OP10B_RH_ROTY(
	bAxis1_Ref_Switch:= , 
	bInit:= OP10_SRV_BLCK_INTZ , 
	bErrorReset:= Servo_Reset, 
	bEnable:= Servo_Enable , 
	bMoveVelocity:= , 
	bHalt:= , 
	bManualMode:= OP10B_MANUAL_SELECTED , 
	fHomePos:= , 
	fOverride:= , 
	fTargetPosition:= OP10B_SRV_RH_BDYANG_CNT.Position, 
	fTargetVelocity:= OP10_SERVO_POS_VEL_LIMIT.OP10B_RH_ROTRY_VELOCITY, 
	fAcc:= , 
	fDec:= , 
	Servo_High_Limit:= OP10_SERVO_POS_VEL_LIMIT.OP10B_RH_ROTRY_POS_LIMIT,
    Servo_Low_Limit:=OP10_SERVO_POS_VEL_LIMIT.OP10B_RH_ROTRY_NEG_LIMIT, 
	Safe_move_Conditions:= Servo_Safety,
	TORQUE_APPLIED :=  , 
	Axis:= OP10B_RH_ROTARY, 
	bHome:= OP10B_SRV_RH_BDYANG_CNT.Axis_Home_Cmd, 
	bSetPosition:= FESTO_NOT_NEED , 
	bMoveAbsolute:= OP10B_SRV_RH_BDYANG_CNT.ABSmove_Start, 
	bMoveRelative:= NOT_REQ , 
	bMoveTorque:= NOT_REQ , 
	stManualModeAxis:= OP10B_SRV_RH_BDYANG_STUS, 
	sAxisState=> OP10B_SRV_RH_BDYANG_CNT.Axis_State, 
	bAxis_ready=> , 
	bAxisInPosition=> , 
	bAxisError=> OP10B_SRV_RH_BDYANG_CNT.Axis_Error, 
	bAxisEnabled=> , 
	bAxisHomed=> , 
	bSetPositionDone=> , 
	bHaltDone=> , 
	bSTOPDone=> , 
	bHomeDone=> OP10B_SRV_RH_BDYANG_CNT.Axis_In_Home, 
	bDone=> , 
	bTorqueReached=> , 
	bsafe_to_move=> , 
	baxis_in_home_pos=> , 
	bABS_Pos_done=> OP10B_SRV_RH_BDYANG_CNT.Axis_In_Pos, 
	Actual_position=>,
	Actual_velocity=> , 
	Actual_Torque=> );
	
OP10B_LH_GRIPR(
	bAxis1_Ref_Switch:= , 
	bInit:= OP10_SRV_BLCK_INTZ , 
	bErrorReset:= Servo_Reset, 
	bEnable:= Servo_Enable , 
	bMoveVelocity:= , 
	bHalt:= , 
	bManualMode:= OP10B_MANUAL_SELECTED , 
	fHomePos:= , 
	fOverride:= , 
	fTargetPosition:= OP10B_SRV_LH_BDYGRP_CNT.Position, 
	fTargetVelocity:= OP10_SERVO_POS_VEL_LIMIT.OP10B_LH_GRPR_VELOCITY, 
	fAcc:= , 
	fDec:= ,
	Servo_High_Limit:= OP10_SERVO_POS_VEL_LIMIT.OP10B_LH_GRPR_POS_LIMIT,
    Servo_Low_Limit:=OP10_SERVO_POS_VEL_LIMIT.OP10B_LH_GRPR_NEG_LIMIT,  
	Safe_move_Conditions:= Servo_Safety,
	TORQUE_APPLIED := , 
	Axis:= OP10B_LH_GRIPPER, 
	bHome:= OP10B_SRV_LH_BDYGRP_CNT.Axis_Home_Cmd, 
	bSetPosition:= FESTO_NOT_NEED , 
	bMoveAbsolute:= OP10B_SRV_LH_BDYGRP_CNT.ABSmove_Start, 
	bMoveRelative:= NOT_REQ , 
	bMoveTorque:= NOT_REQ , 
	stManualModeAxis:= OP10B_SRV_LH_BDYGRP_STUS, 
 	sAxisState=> OP10B_SRV_LH_BDYGRP_CNT.Axis_State, 
	bAxis_ready=> , 
	bAxisInPosition=> , 
	bAxisError=> OP10B_SRV_LH_BDYGRP_CNT.Axis_Error, 
	bAxisEnabled=> , 
	bAxisHomed=> , 
	bSetPositionDone=> , 
	bHaltDone=> , 
	bSTOPDone=> , 
	bHomeDone=> OP10B_SRV_LH_BDYGRP_CNT.Axis_In_Home, 
	bDone=> , 
	bTorqueReached=> , 
	bsafe_to_move=> , 
	baxis_in_home_pos=> , 
	bABS_Pos_done=> OP10B_SRV_LH_BDYGRP_CNT.Axis_In_Pos , 
	Actual_position=>, 
	Actual_velocity=> , 
	Actual_Torque=> );
	
OP10B_RH_GRIPR(
	bAxis1_Ref_Switch:= , 
	bInit:= OP10_SRV_BLCK_INTZ , 
	bErrorReset:= Servo_Reset, 
	bEnable:= Servo_Enable  , 
	bMoveVelocity:= , 
	bHalt:= , 
	bManualMode:= OP10B_MANUAL_SELECTED , 
	fHomePos:= , 
	fOverride:= , 
	fTargetPosition:= OP10B_SRV_RH_BDYGRP_CNT.Position, 
	fTargetVelocity:= OP10_SERVO_POS_VEL_LIMIT.OP10B_RH_GRPR_VELOCITY, 
	fAcc:= , 
	fDec:= ,
	Servo_High_Limit:= OP10_SERVO_POS_VEL_LIMIT.OP10B_RH_GRPR_POS_LIMIT,
    Servo_Low_Limit:=OP10_SERVO_POS_VEL_LIMIT.OP10B_RH_GRPR_NEG_LIMIT, 
	Safe_move_Conditions:=Servo_Safety,
	TORQUE_APPLIED := , 
	Axis:= OP10B_RH_GRIPPER, 
	bHome:= OP10B_SRV_RH_BDYGRP_CNT.Axis_Home_Cmd, 
	bSetPosition:= FESTO_NOT_NEED , 
	bMoveAbsolute:= OP10B_SRV_RH_BDYGRP_CNT.ABSmove_Start, 
	bMoveRelative:= NOT_REQ , 
	bMoveTorque:= NOT_REQ , 
	stManualModeAxis:= OP10B_SRV_RH_BDYGRP_STUS, 
 	sAxisState=> OP10B_SRV_RH_BDYGRP_CNT.Axis_State, 
	bAxis_ready=> , 
	bAxisInPosition=>, 
	bAxisError=> OP10B_SRV_RH_BDYGRP_CNT.Axis_Error, 
	bAxisEnabled=> , 
	bAxisHomed=> , 
	bSetPositionDone=> , 
	bHaltDone=> , 
	bSTOPDone=> , 
	bHomeDone=> OP10B_SRV_RH_BDYGRP_CNT.Axis_In_Home,  
	bDone=> , 
	bTorqueReached=> , 
	bsafe_to_move=> , 
	baxis_in_home_pos=> , 
	bABS_Pos_done=>  OP10B_SRV_RH_BDYGRP_CNT.Axis_In_Pos , 
	Actual_position=>, 
	Actual_velocity=> , 
	Actual_Torque=> );
	
	
OP10B_CONVEYOR(
	bAxis1_Ref_Switch:= , 
	bInit:= , 
	bErrorReset:= Servo_Reset , 
	bEnable:= Servo_Enable, 
	bMoveVelocity:=OP10B_SRV_O_CNVY_CNT.VELmove_Start, 
	bHalt:= , 
	bManualMode:= OP10B_MANUAL_SELECTED, 
	fHomePos:= , 
	fOverride:= , 
	fTargetPosition:=OP10B_SRV_O_CNVY_CNT.Position , 
	fTargetVelocity:=OP10B_SRV_O_CNVY_CNT.Velocity , 
	fAcc:= , 
	fDec:= , 
	Safe_move_Conditions:= Servo_Safety, 
	Axis:= OP10B_CONVRY, 
	HME_WRITE_ADD:= 16#5003,	
	bHome:= OP10B_SRV_O_CNVY_CNT.Bsethome , 
	bSetPosition:= OP10B_SRV_O_CNVY_CNT.BsetPos, 
	bMoveAbsolute:= OP10B_SRV_O_CNVY_CNT.ABSmove_Start, 
	bMoveRelative:= OP10B_SRV_O_CNVY_CNT.RELmove_Start, 
	bMoveTorque:= OP10B_SRV_O_CNVY_CNT.Torque_mode_Start, 
	stManualModeAxis:= OP10B_SRV_O_CNVY_STUS, 
	bmove_home:= OP10B_SRV_O_CNVY_CNT.Axis_Home_Cmd, 
	sAxisState=>OP10B_SRV_O_CNVY_CNT.Axis_State , 
	bAxis_ready=>OP10B_SRV_O_CNVY_CNT.Axis_ready , 
	bAxisInPosition=> , 
	bAxisError=> OP10B_SRV_O_CNVY_CNT.Axis_Error, 
	bAxisEnabled=> , 
	bAxisHomed=> , 
	bSetPositionDone=> , 
	bHaltDone=> , 
	bSTOPDone=> , 
	bHomeDone=> OP10B_SRV_O_CNVY_CNT.Axis_In_Home, 
	bDone=> , 
	bTorqueReached=> , 
	bsafe_to_move=> , 
	baxis_in_home_pos=> , 
	bABS_Pos_done=> , 
	Actual_position=> , 
	Actual_velocity=> , 
	Actual_Torque=> );
	
	   OP10A_SRV_RH_BDYANG_STUS.targetVelocity	:= 20;//OP10A_TARGET_VEL	
	   OP10A_SRV_LH_BDYANG_STUS.targetVelocity	:= 20;//OP10A_TARGET_VEL	
	   OP10A_SRV_RH_BDYGRP_STUS.targetVelocity	:= 20;//OP10A_TARGET_VEL	
	   OP10A_SRV_LH_BDYGRP_STUS.targetVelocity	:= 20;//OP10A_TARGET_VEL	
	   OP10A_SRV_LH_BDYGRP_STUS.targetVelocity	:= 20;//OP10A_TARGET_VEL	
	
	   OP10B_SRV_RH_BDYANG_STUS.targetVelocity	:= 20;//OP10B_TARGET_VEL	
	   OP10B_SRV_LH_BDYANG_STUS.targetVelocity	:= 20;//OP10B_TARGET_VEL	
	   OP10B_SRV_RH_BDYGRP_STUS.targetVelocity	:= 20;//OP10B_TARGET_VEL	
	   OP10B_SRV_LH_BDYGRP_STUS.targetVelocity	:= 20;//OP10B_TARGET_VEL	
	   OP10B_SRV_LH_BDYGRP_STUS.targetVelocity	:= 20;//OP10B_TARGET_VEL	
	
	
		OP10_SRV_FRST_PCKBDY_STUS.TARgetVelocity:=50;
		OP10_SRV_SCND_PCKBDY_STUS.TARgetVelocity:=50;

END_PROGRAM

// ---- FB/In_Range.TcPOU
FUNCTION In_Range : BOOL
VAR_INPUT
	value,setvalue,tolerance:LREAL;
END_VAR
VAR
	low: LREAL:= setvalue-tolerance;
	high:LREAL:= setvalue+tolerance;;
END_VAR

IF (value>=low) AND (value<=high) THEN
	In_Range:=TRUE;
ELSE
	In_Range:=FALSE;
END_IF

END_FUNCTION

// ---- POUs/Programs/OP10/OP10_HOMING.TcPOU
PROGRAM OP10_HOMING
VAR
	OP10A_ERR_TMR				: TON;
	OP10B_ERR_TMR				: TON;
	OP10A_ROBO_RST_SEQ			: INT;	
	OP10B_ROBO_RST_SEQ			: INT;
	OP10A_START_HOMING			: BOOL;
	OP10B_START_HOMING			: BOOL;
	OP10A_ROBO_INZI_DN			: BOOL;	
	OP10B_ROBO_INZI_DN			: BOOL;	
	temp_42						: BOOL;	
	temp_43						: BOOL;	
END_VAR

//#############################		OP10	###########################################

IF (OP10A_START_HOMNG OR OP10B_START_HOMNG) AND (NOT (OP10A_AUTO_RUNNING OR OP10A_STEP_RUNNING OR OP10B_AUTO_RUNNING OR OP10B_STEP_RUNNING OR 
	 OP10A_Rbt_In_Pick_Zone OR OP10B_Rbt_In_Pick_Zone)) THEN
	OP10_A_SRV_SCND_BDYPCK_HME		:= (OP10_BDY_SING_FRT.Sensor1 AND OP10_BDY_SING_SEC.Sensor1) OR OP10_COMP_PICKED_1;		
	OP10_A_SRV_FST_BDYPCK_HME	    := (OP10_BDY_SING_FRT.Sensor1 AND OP10_BDY_SING_SEC.Sensor1) OR OP10_COMP_PICKED_2;
	OP10_FRT_CYL_INITZAL			:= NOT OP10_COMP_PICKED_1;
	OP10_SEC_CYL_INITZAL			:= NOT OP10_COMP_PICKED_2;	
END_IF

//#############################		OP10A	################################

R1(CLK:= OP10A_START_HOMING AND NOT OP10A_ERR AND NOT OP10A_AUTO_RUNNING AND NOT OP10A_STEP_RUNNING, Q=> );
IF R1.Q THEN
	OP10A_START_HOMNG		:= TRUE;
	OP10A_START_HOMING		:= FALSE;
	OP10A_HME_STP_NO		:= 1;
	OP10A_ROBO_RST_SEQ		:= 0;
	OP10_COMP_PICKED_1		:= 0;	// need to be deleted
	OP10_COMP_PICKED_2		:= 0;
	OP10A_Sing_Seq			:=10;
	OP10B_Sing_Seq			:=10;	
END_IF
IF OP10A_ALL_HOME OR OP10A_ERR THEN
	OP10A_START_HOMNG		:= FALSE;	
END_IF

IF (OP10A_HME_STP_NO = 10) AND OP10A_START_HOMNG THEN
	OP10A_ROBO_SFE_HME		:= TRUE;
IF OP10A_Rbt_In_Home THEN
	OP10A_HME_STP_NO 		:= OP10A_HME_10_15;
END_IF
END_IF

OP10A_ALL_HOME	:= OP10_SRV_FRST_PCKBDY_HME_FB AND OP10_SRV_SCND_PCKBDY_HME_FB AND OP10A_Rbt_In_Home AND 
					(OP10A_HME_STP_NO=30)AND (OP10A_ROBO_RST_SEQ=30) AND OP10A_GRIPPER_HOME AND ((OP10_BDY_SING_FRT.Sensor1 OR OP10_COMP_PICKED_1)AND 
						(OP10_BDY_SING_SEC.Sensor1 OR OP10_COMP_PICKED_2));



//####################################		OP10A_ROBO	RST		#################################

IF OP10A_START_HOMNG THEN
CASE OP10A_ROBO_RST_SEQ OF 
	
	0: 	OP10A_ROBO_MODE_NO				:= 3;	
		OP10A_ROBO_PRGM_RST				:= TRUE;
		OP10A_ROBO_RST_SEQ				:= 5;
		
	5:	IF (OP10A_ROBO_PRGM_RST =TRUE) AND (NOT OP10A_Program_Execute) THEN
		IF NOT OP10A_CMP_PRS_ROBO THEN
		OP10A_Homing_Start				:= TRUE;
		OP10A_ROBO_RST_SEQ				:= 10;
		ELSE
		OP10A_Homing_Start				:= TRUE;
		OP10A_PLACE_IN_REJECTION		:= TRUE;
		OP10A_ROBO_RST_SEQ				:= 100;	
		END_IF		
		OP10A_ROBO_PRGM_RST				:= FALSE;		
		END_IF	
	
	10: IF OP10A_Rbt_In_Home THEN
		OP10A_Homing_Start				:= FALSE;
		OP10A_ROBO_RST_SEQ				:= 15;
		END_IF

	15: IF OP10A_Rbt_In_Home THEN
		OP10A_Homing_Start				:= FALSE;
		OP10A_ROBO_MODE_NO				:= 1;
		OP10A_ROBO_PRGM_RST				:= TRUE;
		OP10A_ROBO_RST_SEQ				:= 20;			
		END_IF

	20: IF (OP10A_ROBO_MODE_NO=1) AND OP10A_ROBO_PRGM_RST AND NOT OP10A_Program_Execute THEN
		OP10A_ROBO_PRGM_RST				:= FALSE;
		OP10A_ROBO_RST_SEQ				:= 30;		
		END_IF

	100: IF OP10A_Rbt_In_Reject_Zone AND OP10A_ROBO_Gripper_Open THEN
		OP10A_PLACE_IN_REJECTION		:= FALSE;
		OP10A_ROBO_RST_SEQ				:= 15;
		 END_IF
END_CASE
END_IF

//#############################		OP10B	################################

R2(CLK:= OP10B_START_HOMING AND NOT OP10B_ERR AND NOT OP10B_AUTO_RUNNING AND NOT OP10B_STEP_RUNNING, Q=> );
IF R2.Q THEN
	OP10B_START_HOMNG		:= TRUE;
	OP10B_START_HOMING		:= FALSE;
	OP10B_HME_STP_NO		:= 1;
	OP10B_ROBO_RST_SEQ		:= 0;
	OP10_COMP_PICKED_1		:= 0;	// need to be deleted
	OP10_COMP_PICKED_2		:= 0;
	OP10A_Sing_Seq			:=10;
	OP10B_Sing_Seq			:=10;	
END_IF
IF OP10B_ALL_HOME OR OP10B_ERR THEN
	OP10B_START_HOMNG		:= FALSE;	
END_IF

IF (OP10B_HME_STP_NO = 10) AND OP10B_START_HOMNG THEN
	OP10B_ROBO_SFE_HME	:= TRUE;
IF OP10B_Rbt_In_Home THEN
	OP10B_HME_STP_NO := OP10B_HME_10_15;
END_IF
END_IF

OP10B_ALL_HOME	:= OP10_SRV_FRST_PCKBDY_HME_FB AND OP10_SRV_SCND_PCKBDY_HME_FB AND OP10B_Rbt_In_Home AND 
					(OP10B_HME_STP_NO=30) AND (OP10B_ROBO_RST_SEQ=30)AND OP10B_GRIPPER_HOME AND ((OP10_BDY_SING_FRT.Sensor1 OR OP10_COMP_PICKED_1)AND 
						(OP10_BDY_SING_SEC.Sensor1 OR OP10_COMP_PICKED_2)); 



//####################################		OP10B_ROBO	RST		#################################

IF OP10B_START_HOMNG THEN
CASE OP10B_ROBO_RST_SEQ OF 
	
	0:	OP10B_ROBO_MODE_NO				:= 3;	
		OP10B_ROBO_PRGM_RST				:= TRUE;
		OP10B_ROBO_RST_SEQ				:= 5;
		
	5:	IF (OP10B_ROBO_PRGM_RST =TRUE) AND (NOT OP10B_Program_Execute) THEN
		IF NOT OP10B_CMP_PRS_ROBO THEN
		OP10B_Homing_Start				:= TRUE;
		OP10B_ROBO_RST_SEQ				:= 10;
		ELSE
		OP10B_Homing_Start				:= TRUE;
		OP10B_PLACE_IN_REJECTION		:= TRUE;
		OP10B_ROBO_RST_SEQ				:= 100;	
		END_IF		
		OP10B_ROBO_PRGM_RST				:= FALSE;		
		END_IF	
	
	10: IF OP10B_Rbt_In_Home THEN
		OP10B_Homing_Start				:= FALSE;
		OP10B_ROBO_RST_SEQ				:= 15;
		END_IF

	15: IF OP10B_Rbt_In_Home THEN
		OP10B_Homing_Start				:= FALSE;
		OP10B_ROBO_MODE_NO				:= 1;
		OP10B_ROBO_PRGM_RST				:= TRUE;
		OP10B_ROBO_RST_SEQ				:= 20;			
		END_IF

	20: IF (OP10B_ROBO_MODE_NO=1) AND OP10B_ROBO_PRGM_RST AND NOT OP10B_Program_Execute THEN
		OP10B_ROBO_PRGM_RST				:= FALSE;
		OP10B_ROBO_RST_SEQ				:= 30;		
		END_IF

	100: IF OP10B_Rbt_In_Reject_Zone AND OP10B_ROBO_Gripper_Open THEN
		OP10B_PLACE_IN_REJECTION		:= FALSE;
		OP10B_ROBO_RST_SEQ				:= 15;
		 END_IF
END_CASE	
END_IF

END_PROGRAM

// ---- POUs/Programs/OP10/OP10A_AUTO.TcPOU
PROGRAM OP10A_AUTO
VAR	
	OP10A_ROBO_SYSTEM				: FB_Robot;
	OP10A_CYL_IP					: OP10_ORNG_CYL_IP;
	OP10A_CYL_OP					: OP10_ORNG_CYL_OP;
	OP10A_PNP_FB					: OP10_ORING_PNP;
	OP10A_ROBO_PNP_FB				: OP10_ROBO_PNP;
	OP10A_STN_MOVER					: INT;
	OP10A_OUT_ORNG_DN				: BOOL;
	OP10A_AGLE_LH_CMR_TRG			: BOOL;
	OP10A_AGLE_RH_CMR_TRG			: BOOL;	
	OP10A_RDY_TO_PLC_ORNG			: BOOL;
	OP10A_STN_ENABLE				: BOOL;
// TEMPERY


	OP10A_ROBO_MANUAL: BOOL;
	ORING_DN: BOOL;
	tmr: Ton;
	OP10A_PROCESS_DN: BOOL;
	OP10A_PROCESS_DN_: BOOL;
	
	OP10A_PROCESS_DN_TRG: R_TRIG;
	

END_VAR

VAR PERSISTENT
	OP10A_RESULT_UPDATE		: INT;
	OP10A_DELAY_TMR			: OP10_ORNG_CYL_DLY;
AFT_DEG_HME_DLY: TIME;	AFT_DEG_WRK_DLY: TIME;
	AFT_GRP_HME_DLY: TIME;
	AFT_GRP_WRK_DELY: TIME;
	AFT_HORZ_FRW_DELY: TIME;
END_VAR

OP10A_PNP_FB(
	AUTO:= OP10A_AUTO_RUNNING OR OP10A_STEP_RUNNING, 
	MANUAL:= OP10A_MANUAL_SELECTED, 
	ERROR:= OP10A_ERR, 
	START_ENABLE:= OP10A_START_ENABLE, 
	ROBO_MVED_SFE:= NOT OP10A_Rbt_In_O_Ring_Zone, 
	LH_CMR_OK:= OP10A_LH_CMR_OK AND OP10A_ORNG_RDY_PCK, 
	LH_CMR_NOK:= OP10A_LH_CMR_NOK AND OP10A_ORNG_RDY_PCK, 
	RH_CMR_OK:= OP10A_RH_CMR_OK AND OP10A_ORNG_RDY_PCK, 
	RH_CMR_NOK:= OP10A_RH_CMR_NOK AND OP10A_ORNG_RDY_PCK, 
	ROBO_REACHED:= OP10A_RDY_TO_PLC_ORNG, 
	CYL_INPUTS:= OP10A_CYL_IP, 
	DELY_TIME:= OP10A_DELAY_TMR,
	CONTINOUS_CHECK := OP10A_CYL_PNP_CHECK, 
	O_RING_PLCED=> OP10A_OUT_ORNG_DN, 
	RDY_TO_PICK_ORNG=> OP10A_CYL_RDY_TO_PLC, 
	LH_REJ_DONE=> , 
	RH_REJ_DONE=> , 
	CYL_OUTPUTS=> OP10A_CYL_OP,
	ORNG_PCK_FRM_CNVY := OP10A_ORNG_PCK_DN);

	
	
	
// OP10A AUTO LOGIC CYLINDERS MAPPING 

									(*SENSOR_I/P*)
	OP10A_CYL_IP.DEGREE_0				:=I10A_ORING_ROTRY_CYL_O_DEG_I1011_0;
	OP10A_CYL_IP.DEGREE_180				:=I10A_ORING_ROTRY_CYL_180_DEG_I1011_1;
    OP10A_CYL_IP.HORIZ_CYL_SNR1         :=I10A_ORING_HORZ_CYL_REV_I1011_2;
    OP10A_CYL_IP.HORIZ_CYL_SNR2         :=I10A_ORING_HORZ_CYL_FWD_I1011_3;
    OP10A_CYL_IP.LH_O_GRP_SNR1       	:=I10A_ORING_LH_GRPR_CLSE_I1010_2;
    OP10A_CYL_IP.LH_O_GRP_SNR2          :=I10A_ORING_LH_GRPR_OPN_I1010_3; 
    OP10A_CYL_IP.LH_O_PUSH_SNR1         := NOT I10A_ORING_LH_PUSHR_CYL_REV_I1010_4;
    OP10A_CYL_IP.LH_O_PUSH_SNR2         :=I10A_ORING_LH_PUSHR_CYL_REV_I1010_4;
    OP10A_CYL_IP.LH_REJ_SNR1            :=I10A_LH_FIRTRE_ORING_REJ_CYL_REV_I1011_6;
    OP10A_CYL_IP.LH_REJ_SNR2            :=I10A_LH_FIRTRE_ORING_REJ_CYL_FWD_I1011_7;
	OP10A_CYL_IP.RH_O_GRP_SNR1			:=I10A_ORING_RH_GRPR_CLSE_I1010_6;
    OP10A_CYL_IP.RH_O_GRP_SNR2          :=I10A_ORING_RH_GRPR_OPN_I1010_5;
    OP10A_CYL_IP.RH_O_PUSH_SNR1         := NOT I10A_ORING_RH_PUSHR_CYL_REV_I1010_7;
    OP10A_CYL_IP.RH_O_PUSH_SNR2         :=I10A_ORING_RH_PUSHR_CYL_REV_I1010_7;
    OP10A_CYL_IP.RH_REJ_SNR1            :=I10A_RH_FIRTRE_ORING_REJ_CYL_REV_I1020_0;
    OP10A_CYL_IP.RH_REJ_SNR2            :=I10A_RH_FIRTRE_ORING_REJ_CYL_FWD_I1020_1;
    OP10A_CYL_IP.VERT_CYL_SNR1          :=I10A_ORING_VERT_CYL_UP_I1011_4;
    OP10A_CYL_IP.VERT_CYL_SNR2          :=I10A_ORING_VERT_CYL_DWN_I1011_5;
	
									(*CYLINDER_AUTO_O/P*)	
	
	OP10A_ALL_CYL_HOME_FB				:=OP10A_CYL_OP.ALL_HOME			  ;
	OP10A_O_0DEGRE_AUTOCMD1				:=OP10A_CYL_OP.DEGREE_AUT_CMD1	  ;
	OP10A_O_180DEGRE_AUTOCMD2   		:=OP10A_CYL_OP.DEGREE_AUT_CMD2    ;
	OP10A_O_HORZ_AUTOCMD1    			:=OP10A_CYL_OP.HORIZ_CYL_AUT_CMD1 ;
	OP10A_O_HORZ_AUTOCMD2    			:=OP10A_CYL_OP.HORIZ_CYL_AUT_CMD2 ;
	OP10A_A_O_LHGRIP_ONOFF    			:=OP10A_CYL_OP.LH_O_GRP_VALVE_ON  ;
	OP10A_A_O_LHPUSH_CYL    			:=OP10A_CYL_OP.LH_O_PSH_VALVE_ON  ;
	OP10A_A_O_RHGRIP_ONOFF    			:=OP10A_CYL_OP.RH_O_GRP_VALVE_ON  ;
	OP10A_A_O_RHPUSH_CYL    			:=OP10A_CYL_OP.RH_O_PSH_VALVE_ON  ;
	OP10A_O_VERT_AUTOCMD1    			:=OP10A_CYL_OP.VERT_CYL_AUT_CMD1  ;
	OP10A_O_VERT_AUTOCMD2    			:=OP10A_CYL_OP.VERT_CYL_AUT_CMD2  ;

// 								DELAY_TIMER_FOR_CYLINDER

	OP10A_DELAY_TMR.AFT_DEG_HME_DLY		:= AFT_DEG_HME_DLY;
	OP10A_DELAY_TMR.AFT_DEG_WRK_DLY		:= AFT_DEG_WRK_DLY;
	OP10A_DELAY_TMR.AFT_GRP_HME_DLY		:= AFT_GRP_HME_DLY;
	OP10A_DELAY_TMR.AFT_GRP_WRK_DELY	:= AFT_GRP_WRK_DELY;
	OP10A_DELAY_TMR.AFT_HORZ_FRW_DELY	:= AFT_HORZ_FRW_DELY;
	







	
	
//###############		ROBO	################### 

OP10A_ROBO_PNP_FB(
	AUTO:= OP10A_AUTO_RUNNING OR OP10A_STEP_RUNNING, 
	MANUAL:= OP10A_MANUAL_SELECTED, 
	ERROR:= OP10A_ERR, 
	START_ENABLE:= OP10A_START_ENABLE, 
	ROBO_STATUS_FB:= OP10A_ROBO_STATUS, 
	ROBO_GRP_STUS:= OP10A_GRP_STATUS, 
	BDY1_RDY_PCK:= OP10_LH_CMP_RDY_PCK, 
	BDY2_RDY_PCK:= OP10_RH_CMP_RDY_PCK, 
	BDY1_PCK_BYPAS:= OP10A_BDY1_PCK_BYPAS, 
	BDY2_PCK_BYPAS:= OP10A_BDY2_PCK_BYPAS, 
	O_RNG_NEED:= , 
	PLC_OUTR_ORNG_DN:= OP10A_OUT_ORNG_DN OR ORING_DN, // DELETE ORING_DN
	CMR_RESULT_DN:= OP10A_CMR_DN_RSLT, 
	LH_CMR_ORNG_OK:= OP10A_LH_CMR_OK, 
	RH_CMR_ORING_OK:= OP10A_RH_CMR_OK,
	STN_ENABLE := OP10A_STN_ENABLE,
	OP10_STN_MOVER := OP10A_STN_MOVER,
	START_HOMING := OP10A_START_HOMNG,
	ROBO_IN_HOME := OP10A_Rbt_In_Home,
	STN_MOVER_NUM := OP10A_STN_MOVER,
	LH_BODY_GRIP_HME_DN := OP10A_SRV_LH_BDYGRP_CNT.Axis_In_Home,
	RH_BODY_GRIP_HME_DN := OP10A_SRV_RH_BDYGRP_CNT.Axis_In_Home,
	LH_BODY_ROTRY_HME_DN := OP10A_SRV_LH_BDYANG_CNT.Axis_In_Home,
	RH_BODY_ROTRY_HME_DN := OP10A_SRV_RH_BDYANG_CNT.Axis_In_Home,
	SEC_SING_CYL_SNR1 := OP10_BDY_SING_SEC.Sensor1,
	FRT_SING_CYL_SNR1 := OP10_BDY_SING_FRT.Sensor1,
	CMP_GRIPPED := OP10A_CMP_PRS_ROBO,
	ROBO_GRP_OPN := OP10A_ROBO_Gripper_Open,
	ROBO_IN_ORING_ZONE := OP10A_Rbt_In_O_Ring_Zone,
	ROBO_CTRL_WRD=> OP10A_ROBO_CNTRL, 
	ROBO_GRP_CNTRL=> OP10A_GRP_CNTRL, 
	LH_CAMERA_TRIGGER=> OP10A_AGLE_LH_CMR_TRG, 
	RH_CAMERA_TRIGGER=> OP10A_AGLE_RH_CMR_TRG, 
	PLC_OUTR_ORNG=> OP10A_RDY_TO_PLC_ORNG,
	LH_PART_STATUS => ,
	RH_PART_STATUS => ,
	PROCESS_DONE => ,
	GRIPPER_HOME => OP10A_GRIPPER_HOME,
	OP10_CURR_MOVER => OP10A_CURR_MOVER,
	PROCESS_DONE := OP10A_PROCESS_DN);


	//OP10A_CMR_DN_RSLT			:= TRUE;						// should be deleted
	//OP10A_LH_CMR_OK             := TRUE;						// should be deleted
	//OP10A_RH_CMR_OK             := TRUE;						// should be deleted	


(*tmr(IN:= OP10A_STN_ENABLE, PT:=T#10MS , Q=> , ET=> );
	IF tmr.Q THEN
	IF (MOVER_CMP_STATUS[OP10A_STN_MOVER][1]=0) THEN
	MOVER_CMP_STATUS[OP10A_STN_MOVER][1] := 10;		
	END_IF
	IF (MOVER_CMP_STATUS[OP10A_STN_MOVER][2]=0) THEN
	MOVER_CMP_STATUS[OP10A_STN_MOVER][2] := 10;
	END_IF	
	ALL_STATION_DONE.POSITION_DONE[OP10A_XTS_POS_NO]:= TRUE;
	END_IF*)
	
	CASE OP10A_RESULT_UPDATE OF
		0: IF OP10A_PROCESS_DN THEN
			OP10A_RESULT_UPDATE			:= 5;
		END_IF
		
		5: 	IF OP10A_PROCESS_DN THEN
			IF (MOVER_CMP_STATUS[OP10A_STN_MOVER][1]=0) THEN
			MOVER_CMP_STATUS[OP10A_CURR_MOVER][1] := OP10A_ROBO_PNP_FB.LH_PART_STATUS;		
			END_IF
			IF (MOVER_CMP_STATUS[OP10A_STN_MOVER][2]=0) THEN
			MOVER_CMP_STATUS[OP10A_CURR_MOVER][2] := OP10A_ROBO_PNP_FB.RH_PART_STATUS;
			END_IF		
			IF OP10A_PROCESS_DN AND (OP10A_CURR_MOVER = OP10A_STN_MOVER) AND (MOVER_CMP_STATUS[OP10A_STN_MOVER][1]=10 OR MOVER_CMP_STATUS[OP10A_STN_MOVER][1]=11) AND 
		(MOVER_CMP_STATUS[OP10A_STN_MOVER][2]=10 OR MOVER_CMP_STATUS[OP10A_STN_MOVER][2]=11) THEN
			OP10A_RESULT_UPDATE			:= 10;
			END_IF
			END_IF
	
		10:	STATION_DONE[OP10A_CURR_MOVER][OP10A_XTS_POS_NO]			:= TRUE;
			IF 	MOVER_STP_NO[OP10A_CURR_MOVER]<>((OP10A_XTS_POS_NO*10)+1)THEN
			OP10A_CURR_MOVER											:= 0;	
			OP10A_PROCESS_DN											:= FALSE;
			OP10A_RESULT_UPDATE											:= 15;
			END_IF
			
		15: OP10A_PROCESS_DN_TRG(CLK:= OP10A_PROCESS_DN, Q=> );
			IF OP10A_PROCESS_DN_TRG.Q THEN
			OP10A_RESULT_UPDATE											:= 0;	
			END_IF
	END_CASE
	

(*	IF OP10A_PROCESS_DN OR tmr.Q THEN
	IF (MOVER_CMP_STATUS[OP10A_STN_MOVER][1]=0) THEN
	MOVER_CMP_STATUS[OP10A_CURR_MOVER][1] := OP10A_ROBO_PNP_FB.LH_PART_STATUS;		
	END_IF
	IF (MOVER_CMP_STATUS[OP10A_STN_MOVER][2]=0) THEN
	MOVER_CMP_STATUS[OP10A_CURR_MOVER][2] := OP10A_ROBO_PNP_FB.RH_PART_STATUS;
	END_IF	
	END_IF
	IF OP10A_PROCESS_DN AND (OP10A_CURR_MOVER = OP10A_STN_MOVER) AND (MOVER_CMP_STATUS[OP10A_STN_MOVER][1]=10 OR MOVER_CMP_STATUS[OP10A_STN_MOVER][1]=11) AND 
		(MOVER_CMP_STATUS[OP10A_STN_MOVER][2]=10 OR MOVER_CMP_STATUS[OP10A_STN_MOVER][2]=11) THEN
	STATION_DONE[OP10A_CURR_MOVER][OP10A_XTS_POS_NO]			:= TRUE;
	IF 	MOVER_STP_NO[OP10A_CURR_MOVER]<>((OP10A_XTS_POS_NO*10)+1)THEN
	OP10A_CURR_MOVER											:= 0;	
	OP10A_PROCESS_DN											:= FALSE;	
	END_IF
	END_IF*)
// #############################		OP10A_ROBO_STATUS_CONTROL		#################################
	
	OP10A_ROBO_STATUS.BDY_PCK_POSITION	  		:= OP10A_ROBO_Gripper_Close AND OP10A_Rbt_In_Pick_Zone;//OP10A_Rbt_In_Pick_Zone
//	OP10A_ROBO_STATUS.BDY_S_PCK_POSITION		:= ;
	OP10A_ROBO_STATUS.BDY_CMR_CHK_POS		  	:= OP10A_Camera_Trigger; 							
//	OP10A_ROBO_STATUS.BDY_S_ORNG_POS		   	:= ;
	OP10A_ROBO_STATUS.BDY_ORNG_PLC_POS	  		:= OP10A_O_Ring_Pick_Pos_Reached AND OP10A_Rbt_In_O_Ring_Zone;//OP10A_Rbt_In_O_Ring_Zone
	OP10A_ROBO_STATUS.BDY_MVE_PLC_POS		  	:= OP10A_ROBO_Gripper_Open;//OP10A_Rbt_In_Place_Zone	
	OP10A_ROBO_STATUS.ROBO_SAFE_POS		    	:=  NOT OP10A_Rbt_In_Place_Zone;
	OP10A_ROBO_STATUS.ROBO_REJ_POS				:= OP10A_Rbt_In_Reject_Zone;

	OP10A_A_BODY_READY_TO_PICK					:= 	OP10A_ROBO_CNTRL.BDY_PCK_POSITION	;	
//	                                      	 	:=  OP10A_ROBO_CNTRL.BDY_S_PCK_POSITION;	    
	OP10A_A_PICK_PART_OK                   		:=  OP10A_ROBO_CNTRL.BDY_CMR_CHK_POS		;
//					                      		:= 	OP10A_ROBO_CNTRL.BDY_S_ORNG_POS		;    
	OP10A_A_CAMERA_OK                      		:= 	OP10A_ROBO_CNTRL.BDY_ORNG_PLC_POS OR OP10A_ROBO_CNTRL.BDY_MVE_PLC_POS;    
//	                                       		:= 	OP10A_ROBO_CNTRL.ROBO_SAFE_POS		;    
//	                                       		:= 	OP10A_ROBO_CNTRL.ROBO_REJ_POS		;   


// #############################		OP10A_GRIPPER_STATUS_CONTROL		#################################

	OP10A_GRP_STATUS.LH_BDY_GRP_WRK_FB			:= OP10A_A_SRV_LH_GRPWRK_FB	;
	OP10A_GRP_STATUS.LH_BDY_GRP_HOM_FB		    := OP10A_A_SRV_LH_GRPHME_FB	;
	OP10A_GRP_STATUS.RH_BDY_GRP_WRK_FB		    := OP10A_A_SRV_RH_GRPWRK_FB	;
	OP10A_GRP_STATUS.RH_BDY_GRP_HME_FB		    := OP10A_A_SRV_RH_GRPHME_FB	;
	OP10A_GRP_STATUS.LH_BDY_ROTRY_WRK_FB		:= OP10A_SRV_LH_BDYANG_WRK_FB;
	OP10A_GRP_STATUS.LH_BDY_ROTRY_HOM_FB		:= OP10A_SRV_LH_BDYANG_HME_FB;
	OP10A_GRP_STATUS.RH_BDY_ROTRY_WRK_FB		:= OP10A_SRV_RH_BDYANG_WRK_FB;
	OP10A_GRP_STATUS.RH_BDY_ROTRY_HME_FB		:= OP10A_SRV_RH_BDYANG_HME_FB;
	OP10A_GRP_STATUS.RH_BDY_ROTRY_ZERO_FB		:= OP10A_SRV_RH_BDYANG_ZERO_FB;
	OP10A_GRP_STATUS.LH_BDY_ROTRY_ZERO_FB		:= OP10A_SRV_LH_BDYANG_ZERO_FB;	
	OP10A_GRP_STATUS.RH_BDY_ROTRY_CMR_FB		:= OP10A_SRV_RH_BDYANG_CMR_FB;
	OP10A_GRP_STATUS.RH_BDY_RTRY_FITEE_FB		:= OP10A_SRV_RH_BDYANG_FITRE_FB;
	OP10A_GRP_STATUS.LH_BDY_ROTRY_CMR_FB		:= OP10A_SRV_LH_BDYANG_CMR_FB;	
	OP10A_GRP_STATUS.LH_BDY_RTRY_FITEE_FB		:= OP10A_SRV_LH_BDYANG_FITRE_FB;

	OP10A_A_SRV_LH_GRPWRK						:= OP10A_GRP_CNTRL.LH_BODY_GRIP_WRK	;
	OP10A_A_SRV_LH_GRPHME	        			:= OP10A_GRP_CNTRL.LH_BODY_GRIP_HOM;
	OP10A_A_SRV_RH_GRPWRK	        			:= OP10A_GRP_CNTRL.RH_BODY_GRIP_WRK	;  
	OP10A_A_SRV_RH_GRPHME	        			:= OP10A_GRP_CNTRL.RH_BODY_GRIP_HME	;
	OP10A_SRV_LH_BDYANG_WRK	        			:= OP10A_GRP_CNTRL.LH_BODY_ROTRY_WRK;	
	OP10A_SRV_LH_BDYANG_HME	        			:= OP10A_GRP_CNTRL.LH_BODY_ROTRY_HOM ;	
	OP10A_SRV_RH_BDYANG_WRK	        			:= OP10A_GRP_CNTRL.RH_BODY_ROTRY_WRK;	
	OP10A_SRV_RH_BDYANG_HME	        			:= OP10A_GRP_CNTRL.RH_BODY_ROTRY_HME ;	
	OP10A_SRV_LH_BDYANG_CMR						:= OP10A_GRP_CNTRL.LH_BODY_ROTRY_CMR;
	OP10A_SRV_LH_BDYANG_FITRE					:= OP10A_GRP_CNTRL.LH_BODY_RTRY_FITEE;	
	OP10A_SRV_RH_BDYANG_CMR						:= OP10A_GRP_CNTRL.RH_BODY_ROTRY_CMR;
	OP10A_SRV_RH_BDYANG_FITRE					:= OP10A_GRP_CNTRL.RH_BODY_RTRY_FITEE;
	
// STEPPER_NEGATIVE_HOME_METHOD
	                                               
	OP10A_SRV_LH_BDYGRP_CNT.Axis_Home_Cmd		:= OP10A_GRP_CNTRL.LH_BODY_GRIP_HOMING_1 ; 
	OP10A_SRV_RH_BDYGRP_CNT.Axis_Home_Cmd		:= OP10A_GRP_CNTRL.RH_BODY_GRIP_HOMING_1 ; 
	OP10A_SRV_LH_BDYANG_CNT.Axis_Home_Cmd		:= OP10A_GRP_CNTRL.LH_BODY_ROTRY_HOMING_1; 		
	OP10A_SRV_RH_BDYANG_CNT.Axis_Home_Cmd		:= OP10A_GRP_CNTRL.RH_BODY_ROTRY_HOMING_1; 
	
	
//#####################################	ROBO_FB	####################################


OP10A_ROBO_SYSTEM(
	i_b_Operation_Enable_Feedback:= OP10A_Auto_Operation_Enable, 
	i_b_Auto_Enable_Feedback:= OP10A_Mirror_Auto_enable, 
	i_b_Servo_On_Feedback:= OP10A_Servo_ON_OFF_Status, 
	i_b_Servo_Off_Feedback:= OP10A_Mirror_SRVO_Off, 
	i_b_Error_Feedback:= OP10A_H_Error OR OP10A_L_Error, 
	i_b_Program_Start_Enable_Feedback:= OP10A_Program_Execute, 
	i_b_Robo_Stopping_Feedback:= OP10A_Program_Waiting, 
	i_b_Emergency_Pressed_Feedback:= OP10A_During_EMG_Stop, 
	i_b_Auto_Mode_Feedback:= OP10A_Mirror_Auto_enable, 
	i_b_Reset:= Servo_Reset, 
	i_b_RobotAutoManual:= OP10A_AUTO_SELECTED OR OP10A_STEP_SELECTED OR OP10A_MANUAL_SELECTED, 
	i_b_ProgramReset:= OP10A_ROBO_PRGM_RST, 
	o_b_Operation_Enable_Cmd=> OP10A_Operation_Enable, 
	o_b_Auto_Enable_Cmd=> OP10A_Auto_Enable, 
	o_b_Servo_On_Cmd=> OP10A_Servo_ON, 
	o_b_Servo_Off_Cmd=> OP10A_SERVO_OFF, 
	o_b_Error_Reset_Cmd=> OP10A_ERR_RST, 
	o_b_Program_Reset_Cmd=> OP10A_PRGM_RST, 
	o_b_Program_Start_Cmd=> OP10A_Start, 
	o_b_Program_Stop_Cmd=> OP10A_Stop , 
	o_b_RobotAutoManual=> , 
	o_b_Error=> );	
	
	OP10A_STOP2					:=OP10A_Stop;
	WITH_ORING_VARIIENT			:= TRUE;				// NEED TO BE CHECKED FOR NOT ORING VARIENT 
	

//##############################			ROBO		#####################################

	IF (MANUAL_SELECTED AND OP10A_M_BODY_READY_TO_PICK) OR 
		(OP10A_A_BODY_READY_TO_PICK AND NOT OP10B_BODY_READY_TO_PICK AND NOT OP10B_Rbt_In_Pick_Zone) THEN
		OP10A_BODY_READY_TO_PICK						:= TRUE;// BODY COMPONENT READY;
		OP10A_Pick_Zone_Safe							:= (OP10A_A_SRV_LH_GRPHME_FB OR OP10A_BDY1_PCK_BYPAS) AND 
															(OP10A_A_SRV_RH_GRPHME_FB OR OP10A_BDY2_PCK_BYPAS ) AND 
 																OP10_LH_CMP_RDY_PCK AND OP10_RH_CMP_RDY_PCK; 
	ELSE
		OP10A_BODY_READY_TO_PICK						:= FALSE;
		OP10A_Pick_Zone_Safe							:= FALSE;					
	END_IF

	IF (MANUAL_SELECTED AND OP10A_M_PICK_PART_OK) OR OP10A_A_PICK_PART_OK THEN
		OP10A_PICK_PART_OK								:= TRUE;
		OP10A_A_ORING_INSERTION_DONE					:= TRUE;
		OP10A_Gripper_Rotate_Complete					:= TRUE;
		OP10A_Camera_Zone_Safe							:= TRUE;(*(OP10A_SRV_RH_BDYANG_CMR_FB OR OP10A_BDY2_PCK_BYPAS) AND 
															(OP10A_SRV_LH_BDYANG_CMR_FB OR OP10A_BDY1_PCK_BYPAS);*)
	ELSE
		OP10A_PICK_PART_OK								:= FALSE;
		OP10A_Gripper_Rotate_Complete					:= FALSE;
		OP10A_Camera_Zone_Safe							:= FALSE;
		OP10A_A_ORING_INSERTION_DONE					:= FALSE;		
	END_IF

	IF (MANUAL_SELECTED AND OP10A_M_PICK_PART_NOK) OR OP10A_A_PICK_PART_NOK THEN
		OP10A_PICK_PART_NOK								:= TRUE;
	ELSE
		OP10A_PICK_PART_NOK								:= FALSE;		
	END_IF

	IF (MANUAL_SELECTED AND OP10A_M_CAMERA_OK) OR OP10A_A_CAMERA_OK THEN
		OP10A_READY_TO_INSERT_ORING						:= TRUE;
		OP10A_Place_Zone_Safe							:= (OP10A_SRV_LH_BDYANG_WRK_FB OR OP10A_BDY1_PCK_BYPAS) AND 
															(OP10A_SRV_RH_BDYANG_WRK_FB OR OP10A_BDY2_PCK_BYPAS);
		OP10A_ROTATION_COMPLETE							:= TRUE;
		OP10A_O_Ring_Zone_Safe							:=  (OP10A_SRV_LH_BDYANG_FITRE_FB OR OP10A_BDY1_PCK_BYPAS) AND 
															(OP10A_SRV_RH_BDYANG_FITRE_FB OR OP10A_BDY2_PCK_BYPAS) AND 
																OP10A_CYL_RDY_TO_PLC;
		IF OP10A_ROBO_CNTRL.BDY_MVE_PLC_POS	THEN
		OP10A_A_PLACE_IN_CONVEYOR						:= TRUE;
		END_IF
		
		IF OP10A_Camera_Trigger THEN
		OP10A_CAMERA_OK									:= TRUE;	
		END_IF												
			
	ELSE                                            	
		OP10A_CAMERA_OK									:= FALSE;
		OP10A_READY_TO_INSERT_ORING						:= FALSE;
		OP10A_O_Ring_Zone_Safe							:= FALSE;
		OP10A_Place_Zone_Safe							:= FALSE;
		OP10A_A_PLACE_IN_CONVEYOR						:= FALSE;
		OP10A_ROTATION_COMPLETE							:= FALSE;		
	END_IF

	IF (MANUAL_SELECTED AND OP10A_M_CAMERA_NOK) OR OP10A_A_CAMERA_NOK AND OP10A_Camera_Trigger THEN
		OP10A_CAMERA_NOK								:= TRUE;
	ELSE
		OP10A_CAMERA_NOK								:= FALSE;		
	END_IF	    	 
              
 	IF (MANUAL_SELECTED AND OP10A_M_ORING_INSERTION_DONE) OR OP10A_A_ORING_INSERTION_DONE THEN
		OP10A_ORING_INSERTION_DONE						:= TRUE;
	ELSE
		OP10A_ORING_INSERTION_DONE						:= FALSE;		
	END_IF 
   
  	IF (MANUAL_SELECTED AND OP10A_M_PLACE_IN_CONVEYOR) OR OP10A_A_PLACE_IN_CONVEYOR THEN
		OP10A_PLACE_IN_CONVEYOR							:= TRUE;
	ELSE
		OP10A_PLACE_IN_CONVEYOR							:= FALSE;		
	END_IF
   
	OP10A_GRIPPER_OPEN									:= (OP10A_A_SRV_LH_GRPHME_FB OR OP10A_BDY1_PCK_BYPAS )AND (OP10A_A_SRV_RH_GRPHME_FB OR OP10A_BDY2_PCK_BYPAS) AND NOT OP10A_ROBO_Gripper_Close;
	OP10A_GRIPPER_CLOSE									:= (OP10A_A_SRV_LH_GRPWRK_FB OR OP10A_BDY1_PCK_BYPAS)AND (OP10A_A_SRV_RH_GRPWRK_FB OR OP10A_BDY2_PCK_BYPAS) AND OP10A_ROBO_Gripper_Close;

	OP10A_Reject_Zone_Safe								:= NOT OP10B_Rbt_In_Reject_Zone;








//############################		OP10A STATION ENABLE CONDITION		##########################

	OP10A_STN_MOVER					:= MOVER_POSITION[OP10A_XTS_POS_NO];
	IF AUTO_WITH_XTS THEN	
	IF OP10A_STN_MOVER>0 THEN
	IF NOT END_OF_CYCLE THEN
	OP10A_STN_ENABLE				:= MOVER_POS_RECHED[OP10A_STN_MOVER] AND ((MOVER_CMP_STATUS[OP10A_STN_MOVER][1]=0)OR 
										(MOVER_CMP_STATUS[OP10A_STN_MOVER][2]=0)) AND STATION_ENABLE_CONTROL AND NOT 
											(I10A_BDY1_PRSN_MOVER_I1001_3 OR I10A_BDY2_PRSN_MOVER_I1001_4);
	ELSE
	MOVER_CMP_STATUS[OP10A_STN_MOVER][1]					:=5;
	MOVER_CMP_STATUS[OP10A_STN_MOVER][2]					:=5;
	STATION_DONE[OP10A_STN_MOVER][OP10A_XTS_POS_NO]			:= TRUE;
	
	END_IF
	ELSE
	OP10A_STN_ENABLE										:= FALSE;	
	END_IF	
	END_IF

END_PROGRAM

// ---- FB/Robot/FB_Robot.TcPOU
FUNCTION_BLOCK FB_Robot
VAR_INPUT
	
	i_b_Operation_Enable_Feedback 		: BOOL;				// IO Enabled Feedback		
	i_b_Auto_Enable_Feedback 			: BOOL;				// Auto Enabled Feedback
	i_b_Servo_On_Feedback 				: BOOL;				// Servo On Feedback		
	i_b_Servo_Off_Feedback 				: BOOL;				// Servo Off Feedback		
	i_b_Error_Feedback					: BOOL;				// Error Feedback		
	i_b_Program_Start_Enable_Feedback 	: BOOL;				// Program Start Enable		
	i_b_Robo_Stopping_Feedback 			: BOOL;				// Robo Stopping Feedback		          		 
	i_b_Emergency_Pressed_Feedback 		: BOOL;				// Emergency Pressed Feedback		
	i_b_Auto_Mode_Feedback 				: BOOL;				// Auto Mode Feedback		bRoboAutoManual

	i_b_Reset							: BOOL;
	i_b_RobotAutoManual					: BOOL;
	i_b_ProgramReset					: BOOL;
	
END_VAR
VAR_OUTPUT
	
	o_b_Operation_Enable_Cmd 			: BOOL;				// IO Enable Command
	o_b_Auto_Enable_Cmd					: BOOL;				// Auto Enable Command
	o_b_Servo_On_Cmd					: BOOL;				// Servo On Command		
	o_b_Servo_Off_Cmd					: BOOL;				// Servo Off Command		
	o_b_Error_Reset_Cmd					: BOOL;				// Error Reset Command	
	o_b_Program_Reset_Cmd				: BOOL;				// Program Reset Command
	o_b_Program_Start_Cmd				: BOOL;				// Program Start Command					
	o_b_Program_Stop_Cmd				: BOOL;				// Program Stop Command	
	
	o_b_RobotAutoManual					: BOOL;
	o_b_Error							: BOOL;
END_VAR

VAR

	iState								: E_State_RobotGeneral;
	tonStateTimeOut						: TON;
	tonAutoManual						: ton;
	bRobotAutoManual					: BOOL;
	
	
END_VAR		

VAR_TEMP
	
	bTIN								: BOOL;	
	bTIN2								: BOOL;
	
END_VAR

	// Auto Manual
	o_b_RobotAutoManual:= i_b_Auto_Enable_Feedback AND NOT bRobotAutoManual;

CASE iState OF 
	

E_State_RobotGeneral.Init:

		o_b_Operation_Enable_Cmd	:= FALSE;
		o_b_Auto_Enable_Cmd			:= false;
		o_b_Servo_On_Cmd			:= false;
		o_b_Servo_Off_Cmd			:= false;
		o_b_Error_Reset_Cmd			:= false;
		o_b_Program_Reset_Cmd		:= false;
		o_b_Program_Start_Cmd		:= false;
		o_b_Program_Stop_Cmd		:= FALSE;
		
		IF i_b_ProgramReset THEN
			iState:=E_State_RobotGeneral.ProgramReset;
		ELSIF NOT i_b_Auto_Enable_Feedback THEN
			iState:=E_State_RobotGeneral.AutoEnable;	
		END_IF

E_State_RobotGeneral.AutoEnable:

		o_b_Operation_Enable_Cmd	:= FALSE;
		o_b_Auto_Enable_Cmd			:= TRUE;
		o_b_Servo_On_Cmd			:= false;
		o_b_Servo_Off_Cmd			:= false;
		o_b_Error_Reset_Cmd			:= false;
		o_b_Program_Reset_Cmd		:= false;
		o_b_Program_Start_Cmd		:= false;
		o_b_Program_Stop_Cmd		:= FALSE;

		bTIN:= i_b_RobotAutoManual;//TRUE;

		IF i_b_ProgramReset THEN
			iState:=E_State_RobotGeneral.ProgramReset;		
		ELSIF i_b_Auto_Enable_Feedback AND i_b_RobotAutoManual THEN
			bTIN:= FALSE;
			iState:=E_State_RobotGeneral.OperationEnable;
		ELSIF tonStateTimeOut.Q THEN 
			bTIN:= FALSE;
			iState:=E_State_RobotGeneral.Init;
		END_IF
		
		tonStateTimeOut(IN:=bTIN,PT:=T#1S);

E_State_RobotGeneral.OperationEnable:

		o_b_Operation_Enable_Cmd	:= TRUE;

		bTIN:= i_b_RobotAutoManual;//TRUE;

		IF i_b_ProgramReset THEN
			iState:=E_State_RobotGeneral.ProgramReset;		
		ELSIF  i_b_Error_Feedback THEN
			bTIN:= FALSE;
			iState:=E_State_RobotGeneral.Error;
		ELSIF NOT i_b_RobotAutoManual THEN
			bTIN:= FALSE;
			iState:=E_State_RobotGeneral.AutoEnable;
		ELSIF i_b_Operation_Enable_Feedback OR i_b_Auto_Enable_Feedback THEN
			bTIN:= FALSE;
			iState:=E_State_RobotGeneral.ServoOn;
		ELSIF tonStateTimeOut.Q THEN 
			bTIN:= FALSE;
			iState:=E_State_RobotGeneral.Error;
		END_IF
		
		tonStateTimeOut(IN:=bTIN,PT:=T#1S);

E_State_RobotGeneral.Error:

		o_b_Operation_Enable_Cmd	:= FALSE;
		o_b_Auto_Enable_Cmd			:= TRUE;
		o_b_Servo_On_Cmd			:= FALSE;
		o_b_Servo_Off_Cmd			:= false;
		o_b_Error_Reset_Cmd			:= false;
		o_b_Program_Reset_Cmd		:= false;
		o_b_Program_Start_Cmd		:= false;
		o_b_Program_Stop_Cmd		:= FALSE;

		IF i_b_ProgramReset THEN
			iState:=E_State_RobotGeneral.ProgramReset;
		ELSIF i_b_reset THEN
		iState:=E_State_RobotGeneral.ErrorReset;	
		END_IF
		
E_State_RobotGeneral.ErrorReset:

		o_b_Auto_Enable_Cmd			:= TRUE;
		o_b_Servo_On_Cmd			:= FALSE;
		o_b_Servo_Off_Cmd			:= false;
		o_b_Error_Reset_Cmd			:= TRUE;
		o_b_Program_Reset_Cmd		:= false;
		o_b_Program_Start_Cmd		:= false;
		o_b_Program_Stop_Cmd		:= FALSE;

		bTIN:= TRUE;

		IF i_b_ProgramReset THEN
			iState:=E_State_RobotGeneral.ProgramReset;		
		ELSIF NOT i_b_Error_Feedback THEN
			bTIN:= FALSE;
			iState:=E_State_RobotGeneral.AutoEnable;	
		ELSIF tonStateTimeOut.Q THEN
			bTIN:= FALSE;
			iState:=E_State_RobotGeneral.Error;
		END_IF

		tonStateTimeOut(IN:=bTIN,PT:=T#1S);

E_State_RobotGeneral.ServoOn:

		o_b_Servo_On_Cmd			:= TRUE;
		
		bTIN:= TRUE;

		IF i_b_ProgramReset THEN
			iState:=E_State_RobotGeneral.ProgramReset;		
		ELSIF  i_b_Error_Feedback THEN
			bTIN:= FALSE;
			iState:=E_State_RobotGeneral.Error;
		ELSIF NOT i_b_RobotAutoManual THEN
			bTIN:= FALSE;
			iState:=E_State_RobotGeneral.AutoEnable;
		ELSIF i_b_Servo_On_Feedback THEN
			bTIN:= FALSE;
			iState:=E_State_RobotGeneral.Start;
		ELSIF tonStateTimeOut.Q THEN	
			bTIN:= FALSE;
			iState:=E_State_RobotGeneral.AutoEnable; // AutoEnable;
		END_IF
		
		tonStateTimeOut(IN:=bTIN,PT:=T#1S);

E_State_RobotGeneral.Start:

		o_b_Program_Start_Cmd		:= TRUE;

		IF i_b_ProgramReset THEN
			iState:=E_State_RobotGeneral.ProgramReset;	
		ELSIF  i_b_Error_Feedback THEN
			iState:=E_State_RobotGeneral.Error;
		ELSIF NOT i_b_RobotAutoManual THEN
			iState:=E_State_RobotGeneral.AutoEnable;
		ELSIF  NOT i_b_Auto_Enable_Feedback OR NOT i_b_Servo_On_Feedback THEN
			iState:=E_State_RobotGeneral.AutoEnable;
		ELSIF i_b_Program_Start_Enable_Feedback THEN
			iState:=E_State_RobotGeneral.Started;
		END_IF
		
E_State_RobotGeneral.Started:

		IF i_b_ProgramReset THEN
			iState:=E_State_RobotGeneral.ProgramReset;	
		ELSIF  i_b_Error_Feedback THEN
			iState:=E_State_RobotGeneral.Error;
		ELSIF NOT i_b_RobotAutoManual THEN
			iState:=E_State_RobotGeneral.AutoEnable;
		ELSIF  NOT i_b_Auto_Enable_Feedback OR NOT i_b_Servo_On_Feedback OR NOT i_b_Program_Start_Enable_Feedback THEN
			iState:=E_State_RobotGeneral.AutoEnable;
		END_IF		
		
E_State_RobotGeneral.ProgramReset: 

		o_b_Operation_Enable_Cmd	:= TRUE;
		o_b_Auto_Enable_Cmd			:= TRUE;
		o_b_Servo_On_Cmd			:= false;
		o_b_Servo_Off_Cmd			:= false;
		o_b_Error_Reset_Cmd			:= TRUE;
		o_b_Program_Reset_Cmd		:= FALSE;
		o_b_Program_Start_Cmd		:= false;
		o_b_Program_Stop_Cmd		:= TRUE;
		
	IF NOT i_b_Error_Feedback THEN
		o_b_Error_Reset_Cmd			:= FALSE;
		o_b_Program_Reset_Cmd			:= TRUE;
	END_IF	
	
		bTIN2:= TRUE;
		
		
	// Auto Manual
		IF tonAutoManual.Q THEN
		bRobotAutoManual:= TRUE;
		END_IF
		
		IF NOT i_b_ProgramReset THEN
			iState:=E_State_RobotGeneral.AutoEnable;
			bTIN2:= FALSE;
			bRobotAutoManual:= FALSE;
		END_IF
		
		

 END_CASE
 tonAutoManual(IN:=bTIN2 , PT:= T#5S , Q=> , ET=> );
 o_b_Error:= (iState=E_State_RobotGeneral.Error) OR (iState=E_State_RobotGeneral.ErrorReset);

END_FUNCTION_BLOCK

// ---- FB/OP10_ORING_PNP.TcPOU
FUNCTION_BLOCK OP10_ORING_PNP
VAR_INPUT
	AUTO					: BOOL;
	MANUAL 					: BOOL;
	ERROR					: BOOL;
	START_ENABLE			: BOOL;
	ROBO_MVED_SFE			: BOOL;
	LH_CMR_OK				: BOOL;
	LH_CMR_NOK				: BOOL;	
	RH_CMR_OK				: BOOL;
	RH_CMR_NOK				: BOOL;
	ROBO_REACHED			: BOOL;	
	CYL_INPUTS				: OP10_ORNG_CYL_IP;
	DELY_TIME				: OP10_ORNG_CYL_DLY;
	CONTINOUS_CHECK: BOOL;
END_VAR
VAR_OUTPUT
	O_RING_PLCED			: BOOL;
	RDY_TO_PICK_ORNG		: BOOL;
	LH_REJ_DONE				: BOOL;
	RH_REJ_DONE				: BOOL;
	CYL_OUTPUTS				: OP10_ORNG_CYL_OP;
END_VAR
VAR
// BOOL
	PNP_CYL_IN_HME			: BOOL;
//INT
	AUTO_STP_NO				: INT;
	LH_REH_STP				: INT;
	RH_REH_STP				: INT;
//TON
	AFT_HORZ_FRWD			: TON;
	AFT_VET_DWN				: TON;
	AFT_GRP_PICK			: TON;
	AFT_DEG_WRK				: TON;
	AFT_GRP_CLS				: TON;
	AFT_PUSH_WRK			: TON;
	AFT_PUSH_HME			: TON;
	AFT_GRP_OPN				: TON;
	
// R_TRIG 
	LH_CAMR_NOK_STRT		: R_TRIG;
	RH_CAMR_NOK_STRT		: R_TRIG;

END_VAR

VAR PERSISTENT
	LH_CMP_GRIPPED			: BOOL;
	RH_CMP_GRIPPED			: BOOL;
END_VAR
VAR_IN_OUT
	ORNG_PCK_FRM_CNVY: BOOL;
END_VAR

IF AUTO OR CONTINOUS_CHECK THEN

IF START_ENABLE OR CONTINOUS_CHECK THEN
		
CASE AUTO_STP_NO OF 
	
		0: IF LH_CMR_OK AND RH_CMR_OK AND NOT LH_CMP_GRIPPED AND NOT RH_CMP_GRIPPED THEN
			AUTO_STP_NO					  :=5;
			END_IF
			IF LH_CMP_GRIPPED AND RH_CMP_GRIPPED THEN
			AUTO_STP_NO					  :=30;		 
			END_IF
			
		5: 	CYL_OUTPUTS.HORIZ_CYL_AUT_CMD1:=FALSE;
			CYL_OUTPUTS.HORIZ_CYL_AUT_CMD2:= TRUE;
			AUTO_STP_NO					  := 10;
					
		10: IF AFT_HORZ_FRWD.Q THEN
			CYL_OUTPUTS.VERT_CYL_AUT_CMD1:=FALSE;
			CYL_OUTPUTS.VERT_CYL_AUT_CMD2:=TRUE;
			AUTO_STP_NO					 := 15;
			END_IF
			
		15: IF AFT_VET_DWN.Q THEN
			IF NOT LH_CMP_GRIPPED THEN
			CYL_OUTPUTS.LH_O_GRP_VALVE_ON:=TRUE;
			LH_CMP_GRIPPED				 :=TRUE;
			END_IF
			IF NOT RH_CMP_GRIPPED THEN
			CYL_OUTPUTS.RH_O_GRP_VALVE_ON:=TRUE;
			RH_CMP_GRIPPED				 :=TRUE;
			END_IF
			AUTO_STP_NO:= 20;
			END_IF
			
		20: IF AFT_GRP_PICK.Q THEN
			CYL_OUTPUTS.VERT_CYL_AUT_CMD2:=FALSE;
			CYL_OUTPUTS.VERT_CYL_AUT_CMD1:=TRUE;
			AUTO_STP_NO					 := 25;
			END_IF
			
		25: IF CYL_INPUTS.VERT_CYL_SNR1 THEN
			ORNG_PCK_FRM_CNVY			:= TRUE;
			CYL_OUTPUTS.HORIZ_CYL_AUT_CMD1:=TRUE;
			CYL_OUTPUTS.HORIZ_CYL_AUT_CMD2:=FALSE;
			AUTO_STP_NO					  := 30;
			END_IF
		
		30: IF CYL_INPUTS.HORIZ_CYL_SNR1 THEN
			CYL_OUTPUTS.LH_O_GRP_VALVE_ON:=TRUE;
			CYL_OUTPUTS.RH_O_GRP_VALVE_ON:=TRUE;
			CYL_OUTPUTS.DEGREE_AUT_CMD2	  := TRUE;
			CYL_OUTPUTS.DEGREE_AUT_CMD1	  := FALSE;
			AUTO_STP_NO					  := 35;			
			END_IF
			
		35: IF AFT_DEG_WRK.Q THEN
			RDY_TO_PICK_ORNG 			  := TRUE;
			AUTO_STP_NO					  := 40;
			END_IF
		
		40: IF ROBO_REACHED OR CONTINOUS_CHECK THEN
			AUTO_STP_NO					  := 45;
			RDY_TO_PICK_ORNG 			  := FALSE;
			END_IF
			
		45: IF AFT_GRP_CLS.Q THEN
			CYL_OUTPUTS.LH_O_PSH_VALVE_ON := TRUE;
			CYL_OUTPUTS.RH_O_PSH_VALVE_ON := TRUE;
			AUTO_STP_NO					  := 50;
			END_IF
		
		50: IF AFT_PUSH_WRK.Q THEN
			O_RING_PLCED				  := TRUE;
			LH_CMP_GRIPPED 				  := FALSE;
			RH_CMP_GRIPPED				  := FALSE;
			CYL_OUTPUTS.LH_O_PSH_VALVE_ON := FALSE;
			CYL_OUTPUTS.RH_O_PSH_VALVE_ON := FALSE;
			AUTO_STP_NO					  := 55;			
			END_IF

		55: IF AFT_PUSH_HME.Q THEN
			AUTO_STP_NO					  := 60;
			END_IF
		
		60: IF AFT_GRP_OPN.Q THEN
			IF ROBO_MVED_SFE OR CONTINOUS_CHECK THEN
			AUTO_STP_NO					  := 65;
			O_RING_PLCED				  := FALSE;	
			END_IF
			END_IF
		
		65: CYL_OUTPUTS.DEGREE_AUT_CMD2	  := FALSE;
			CYL_OUTPUTS.DEGREE_AUT_CMD1	  := TRUE;
			CYL_OUTPUTS.RH_O_GRP_VALVE_ON := FALSE;
			CYL_OUTPUTS.LH_O_GRP_VALVE_ON := FALSE;
			IF CYL_INPUTS.DEGREE_0 THEN				//CYL_INPUTS.RH_O_GRP_SNR1 AND CYL_INPUTS.LH_O_GRP_SNR1 AND 
			AUTO_STP_NO					  := 0;	
			END_IF
			

	
END_CASE

(*////////////////////////LH_REJ/////////////////////////////
LH_CAMR_NOK_STRT(CLK:=LH_CMR_NOK , Q=> );
IF LH_CAMR_NOK_STRT.Q THEN
	 LH_REH_STP							 := 1;
END_IF

CASE LH_REH_STP OF
		
	1: CYL_OUTPUTS.LH_REJ_CMD2			 := TRUE;
	   CYL_OUTPUTS.LH_REJ_CMD1			 := FALSE;
	   LH_REJ_DONE						 := FALSE;
	   LH_REH_STP						 := 5;
	   
	5: IF CYL_INPUTS.LH_REJ_SNR2 THEN
	   CYL_OUTPUTS.LH_REJ_CMD2			 := FALSE;
	   CYL_OUTPUTS.LH_REJ_CMD1			 := TRUE;
	   LH_REH_STP						 := 10;
	   END_IF
	   
	10:IF CYL_INPUTS.LH_REJ_SNR1 THEN
	   LH_REJ_DONE						 := TRUE;
	   LH_REH_STP						 := 15;
	   END_IF     
END_CASE

/////////////////////////////////RH_REJ/////////////////
RH_CAMR_NOK_STRT(CLK:=RH_CMR_NOK , Q=> );
IF RH_CAMR_NOK_STRT.Q THEN
	 RH_REH_STP							 := 1;
END_IF

CASE RH_REH_STP OF
		
	1: CYL_OUTPUTS.RH_REJ_CMD2			 := TRUE;
	   CYL_OUTPUTS.RH_REJ_CMD1			 := FALSE;
	   RH_REJ_DONE						 := FALSE;
	   RH_REH_STP						 := 5;
	   
	5: IF CYL_INPUTS.RH_REJ_SNR2 THEN
	   CYL_OUTPUTS.RH_REJ_CMD2			 := FALSE;
	   CYL_OUTPUTS.RH_REJ_CMD1			 := TRUE;
	   RH_REH_STP						 := 10;
	   END_IF
	   
	10:IF CYL_INPUTS.RH_REJ_SNR1 THEN
	   RH_REJ_DONE						 := TRUE;
	   RH_REH_STP						 := 15;
	   END_IF     
END_CASE*)

END_IF
												(*DELAY_TIMER*)
											
		AFT_HORZ_FRWD(IN:=(AUTO_STP_NO=10 AND CYL_INPUTS.HORIZ_CYL_SNR2) , PT:=(DELY_TIME.AFT_HORZ_FRW_DELY), Q=> , ET=> );
		AFT_VET_DWN(IN:=( AUTO_STP_NO=15 AND CYL_INPUTS.VERT_CYL_SNR2) , PT:=(DELY_TIME.AFT_VERT_DWN_DELY) , Q=> , ET=> );
		AFT_GRP_PICK(IN:=(AUTO_STP_NO=20 AND CYL_INPUTS.LH_O_GRP_SNR2 AND CYL_INPUTS.RH_O_GRP_SNR2) , PT:=(DELY_TIME.AFT_GRP_WRK_DELY) , Q=> , ET=> );
		AFT_DEG_WRK(IN:=(AUTO_STP_NO=35 AND CYL_INPUTS.DEGREE_180) , PT:=(DELY_TIME.AFT_DEG_WRK_DLY) , Q=> , ET=> );
		AFT_GRP_CLS(IN:=(AUTO_STP_NO=45), PT:=(DELY_TIME.AFT_GRP_HME_DLY) , Q=> , ET=> );
		AFT_PUSH_WRK(IN:=(AUTO_STP_NO=50 AND CYL_INPUTS.LH_O_PUSH_SNR2 AND CYL_INPUTS.RH_O_PUSH_SNR2), PT:=(DELY_TIME.AFT_PSH_FRWD_DLY) , Q=> , ET=> );
		AFT_PUSH_HME(IN:=(AUTO_STP_NO=55 AND CYL_INPUTS.LH_O_PUSH_SNR1 AND CYL_INPUTS.RH_O_PUSH_SNR1), PT:=(DELY_TIME.AFT_PSH_REV_DLY) , Q=> , ET=> );
		AFT_GRP_OPN(IN:=(AUTO_STP_NO=60), PT:=(DELY_TIME.AFT_GRP_WRK_DELY) , Q=> , ET=> );
			
ELSE
		
	CYL_OUTPUTS.DEGREE_AUT_CMD1			:= FALSE;
	CYL_OUTPUTS.DEGREE_AUT_CMD2         := FALSE;
	CYL_OUTPUTS.HORIZ_CYL_AUT_CMD1      := FALSE;
	CYL_OUTPUTS.HORIZ_CYL_AUT_CMD2      := FALSE;
	CYL_OUTPUTS.LH_O_GRP_VALVE_ON       := FALSE;
	CYL_OUTPUTS.LH_O_PSH_VALVE_ON       := FALSE;
	CYL_OUTPUTS.RH_O_GRP_VALVE_ON       := FALSE;
	CYL_OUTPUTS.RH_O_PSH_VALVE_ON       := FALSE;
	CYL_OUTPUTS.VERT_CYL_AUT_CMD1       := FALSE;
	CYL_OUTPUTS.VERT_CYL_AUT_CMD2       := FALSE;
	AUTO_STP_NO							:= 0;
	O_RING_PLCED				  		:= FALSE;
	RDY_TO_PICK_ORNG 			 		:= FALSE;	
END_IF

// CYLINDER HOME

IF CYL_INPUTS.DEGREE_0 AND CYL_INPUTS.HORIZ_CYL_SNR1 AND (CYL_INPUTS.LH_O_GRP_SNR1 OR LH_CMP_GRIPPED) AND
	(CYL_INPUTS.RH_O_GRP_SNR1 OR RH_CMP_GRIPPED) AND  CYL_INPUTS.VERT_CYL_SNR1 AND CYL_INPUTS.LH_O_PUSH_SNR1 AND CYL_INPUTS.RH_O_PUSH_SNR1 THEN
	PNP_CYL_IN_HME						 :=TRUE;
	CYL_OUTPUTS.ALL_HOME				 :=TRUE;
ELSE
	CYL_OUTPUTS.ALL_HOME				 :=FALSE;	
	PNP_CYL_IN_HME						 :=FALSE;	
END_IF

END_FUNCTION_BLOCK

// ---- FB/OP10_ROBO_PNP.TcPOU
FUNCTION_BLOCK OP10_ROBO_PNP
VAR_INPUT
	AUTO							: BOOL;
	MANUAL 							: BOOL;
	DRY_RUN							: BOOL;
	ERROR							: BOOL;
	START_ENABLE					: BOOL;
	ROBO_STATUS_FB					: OP10_ROBO_STUS;
	ROBO_GRP_STUS					: OP10_GRP_STATUS;
	BDY1_RDY_PCK					: BOOL;	
	BDY2_RDY_PCK					: BOOL;
	BDY1_PCK_BYPAS 					: BOOL;	
	BDY2_PCK_BYPAS 					: BOOL;
	O_RNG_NEED						: BOOL;
	PLC_OUTR_ORNG_DN				: BOOL;
	CMR_RESULT_DN					: BOOL;
	LH_CMR_ORNG_OK					: BOOL;
	RH_CMR_ORING_OK					: BOOL;
	STN_ENABLE						: BOOL;
	OP10_STN_MOVER					: INT;
	START_HOMING					: BOOL;
	ROBO_IN_HOME					: BOOL;
	STN_MOVER_NUM					: INT;
	LH_BODY_GRIP_HME_DN				: BOOL;
	RH_BODY_GRIP_HME_DN				: BOOL;
	LH_BODY_ROTRY_HME_DN			: BOOL;
	RH_BODY_ROTRY_HME_DN			: BOOL;
	SEC_SING_CYL_SNR1				: BOOL;
	FRT_SING_CYL_SNR1				: BOOL;
	CMP_GRIPPED						: BOOL;
	ROBO_GRP_OPN					: BOOL;
	ROBO_IN_ORING_ZONE				: BOOL;
END_VAR                     		
VAR_OUTPUT                  		
	ROBO_CTRL_WRD					: OP10_ROBO_CNTRL;
	ROBO_GRP_CNTRL					: OP10_GRP_CONTRL;
	LH_CAMERA_TRIGGER				: BOOL;
	RH_CAMERA_TRIGGER				: BOOL;
	PLC_OUTR_ORNG					: BOOL;                       		
	LH_PART_STATUS					: INT;
	RH_PART_STATUS					: INT;
	GRIPPER_HOME					: BOOL;
	OP10_CURR_MOVER					: INT;
END_VAR                     		
VAR 
	LH_GRP							: FB_Axis;
	RH_GRP							: FB_Axis;
	LH_ROTRY						: FB_Axis;
	RH_ROTRY						: FB_Axis; 
	LH_GRP_PULSE					: R_TRIG;
	RH_GRP_PULSE					: R_TRIG;
	RH_ROTRY_PULSE					: R_TRIG;
	LH_ROTRY_PULSE					: R_TRIG;
	LH_GRP_REF						: R_TRIG;
	RH_GRP_REF						: R_TRIG;	
	LH_ROTRY_REF					: R_TRIG;	
	RH_ROTRY_REF					: R_TRIG;
	AUTO_STP_NO						: INT;	
	F_TRE_ANGLE_CHK_DN				: BOOL;
	LH_GRP_HOM_DN					: BOOL;
	RH_GRP_HOM_DN					: BOOL;
	LH_ROTRY_HOM_DN					: BOOL;
	RH_ROTRY_HOM_DN					: BOOL;
	TEMP_3							: BOOL;
	LH_GRP_HME_REF					: BOOL;
	RH_GRP_HME_REF					: BOOL;	
	LH_ROTRY_HME_REF				: BOOL;
	RH_ROTRY_HME_REF				: BOOL;		
	
	CMR_TMR: TON;
END_VAR

VAR PERSISTENT
	O_RNG_CHK_DN					: BOOL;
	OUTER_ORNG_PLC_DN				: BOOL;
END_VAR

VAR_IN_OUT
	PROCESS_DONE					: BOOL;
END_VAR

IF AUTO THEN
IF START_ENABLE THEN
CASE AUTO_STP_NO OF 
	
	0: IF (BDY1_RDY_PCK OR BDY1_PCK_BYPAS) AND (BDY2_RDY_PCK OR BDY2_PCK_BYPAS) AND 
	   		ROBO_STATUS_FB.ROBO_SAFE_POS AND NOT CMP_GRIPPED AND NOT F_TRE_ANGLE_CHK_DN AND
			 NOT OUTER_ORNG_PLC_DN AND NOT O_RNG_CHK_DN THEN
		AUTO_STP_NO						:= 5;
		ROBO_GRP_CNTRL.LH_BODY_ROTRY_HOM:= NOT BDY1_PCK_BYPAS;
		ROBO_GRP_CNTRL.RH_BODY_ROTRY_HME:= NOT BDY2_PCK_BYPAS;
		ROBO_CTRL_WRD.BDY_PCK_POSITION	:= TRUE;
		END_IF
		IF CMP_GRIPPED AND NOT F_TRE_ANGLE_CHK_DN AND NOT ROBO_STATUS_FB.BDY_CMR_CHK_POS AND NOT OUTER_ORNG_PLC_DN AND NOT O_RNG_CHK_DN THEN
		AUTO_STP_NO						:= 15;			
		END_IF
		IF CMP_GRIPPED AND ROBO_STATUS_FB.BDY_CMR_CHK_POS AND NOT OUTER_ORNG_PLC_DN AND NOT O_RNG_CHK_DN THEN
		AUTO_STP_NO						:= 15;				
		END_IF
		IF F_TRE_ANGLE_CHK_DN AND NOT ROBO_STATUS_FB.BDY_CMR_CHK_POS AND NOT OUTER_ORNG_PLC_DN AND NOT O_RNG_CHK_DN THEN
		AUTO_STP_NO						:= 25;			
		END_IF 
		IF OUTER_ORNG_PLC_DN AND NOT O_RNG_CHK_DN THEN
		AUTO_STP_NO						:= 40;			
		END_IF
		IF O_RNG_CHK_DN THEN
		AUTO_STP_NO						:= 50;			
		END_IF		
		
	5: IF ROBO_STATUS_FB.BDY_PCK_POSITION THEN
		ROBO_GRP_CNTRL.LH_BODY_ROTRY_HOM:= FALSE;
		ROBO_GRP_CNTRL.RH_BODY_ROTRY_HME:= FALSE;
		ROBO_CTRL_WRD.BDY_PCK_POSITION	:= FALSE;
		IF NOT BDY1_PCK_BYPAS AND NOT BDY2_PCK_BYPAS THEN
		ROBO_GRP_CNTRL.LH_BODY_GRIP_WRK	:= TRUE;
		ROBO_GRP_CNTRL.RH_BODY_GRIP_WRK	:= TRUE;
		END_IF
		IF BDY1_PCK_BYPAS AND NOT BDY2_PCK_BYPAS THEN
		ROBO_GRP_CNTRL.LH_BODY_GRIP_WRK	:= FALSE;
		ROBO_GRP_CNTRL.RH_BODY_GRIP_WRK	:= TRUE;
		END_IF
		IF NOT BDY1_PCK_BYPAS AND BDY2_PCK_BYPAS THEN
		ROBO_GRP_CNTRL.LH_BODY_GRIP_WRK	:= TRUE;
		ROBO_GRP_CNTRL.RH_BODY_GRIP_WRK	:= FALSE;
		END_IF
		IF ( ROBO_GRP_STUS.LH_BDY_GRP_WRK_FB OR BDY1_PCK_BYPAS) AND ( ROBO_GRP_STUS.RH_BDY_GRP_WRK_FB OR BDY2_PCK_BYPAS) AND 
				FRT_SING_CYL_SNR1 AND SEC_SING_CYL_SNR1 THEN
		AUTO_STP_NO						:= 10;		
		END_IF
		END_IF
		
	10: ROBO_GRP_CNTRL.LH_BODY_GRIP_WRK	:= FALSE;
		ROBO_GRP_CNTRL.RH_BODY_GRIP_WRK	:= FALSE;
		AUTO_STP_NO						:= 15;
		
	15: ROBO_CTRL_WRD.BDY_CMR_CHK_POS	:= TRUE;
		AUTO_STP_NO						:= 16;
		
	16: IF NOT ROBO_STATUS_FB.BDY_PCK_POSITION THEN
		ROBO_GRP_CNTRL.LH_BODY_ROTRY_CMR:= NOT BDY1_PCK_BYPAS;
		ROBO_GRP_CNTRL.RH_BODY_ROTRY_CMR:= NOT BDY2_PCK_BYPAS;
		AUTO_STP_NO						:= 20;
		END_IF

	20: IF ROBO_STATUS_FB.BDY_CMR_CHK_POS THEN
		ROBO_GRP_CNTRL.LH_BODY_ROTRY_CMR:= FALSE;
	    ROBO_GRP_CNTRL.RH_BODY_ROTRY_CMR:= FALSE;
		ROBO_CTRL_WRD.BDY_CMR_CHK_POS	:= FALSE;
		IF NOT BDY1_PCK_BYPAS THEN
		LH_CAMERA_TRIGGER				:= TRUE;
		END_IF
		IF NOT BDY2_PCK_BYPAS THEN
		RH_CAMERA_TRIGGER				:= TRUE;
		END_IF
		IF CMR_RESULT_DN THEN
		AUTO_STP_NO						:= 25;
		END_IF
		END_IF
		
	25: ROBO_CTRL_WRD.BDY_ORNG_PLC_POS	:= TRUE;
		ROBO_GRP_CNTRL.LH_BODY_RTRY_FITEE:= NOT BDY1_PCK_BYPAS;
		ROBO_GRP_CNTRL.RH_BODY_RTRY_FITEE:= NOT BDY2_PCK_BYPAS;
		LH_CAMERA_TRIGGER				:= FALSE;
		RH_CAMERA_TRIGGER				:= FALSE;
		IF (ROBO_GRP_STUS.LH_BDY_RTRY_FITEE_FB OR BDY1_PCK_BYPAS) AND (ROBO_GRP_STUS.RH_BDY_RTRY_FITEE_FB OR BDY2_PCK_BYPAS) THEN
		AUTO_STP_NO						:= 30;
		END_IF
		
	30: ROBO_GRP_CNTRL.RH_BODY_RTRY_FITEE:= FALSE;
		ROBO_GRP_CNTRL.LH_BODY_RTRY_FITEE:= FALSE;
		IF (ROBO_GRP_STUS.LH_BDY_RTRY_FITEE_FB OR BDY1_PCK_BYPAS) AND (ROBO_GRP_STUS.RH_BDY_RTRY_FITEE_FB OR BDY2_PCK_BYPAS) THEN
		F_TRE_ANGLE_CHK_DN				:= TRUE;
		AUTO_STP_NO						:= 35;
		END_IF
//		ROBO_CTRL_WRD.BDY_S_ORNG_POS	:= TRUE;		


	35: IF ROBO_STATUS_FB.BDY_ORNG_PLC_POS THEN
		PLC_OUTR_ORNG					:= TRUE;
		AUTO_STP_NO						:= 40;		
		END_IF
		
	40: IF PLC_OUTR_ORNG_DN THEN
		ROBO_CTRL_WRD.BDY_ORNG_PLC_POS	:= TRUE;
		PLC_OUTR_ORNG					:= FALSE;
		ROBO_CTRL_WRD.BDY_CMR_CHK_POS	:= TRUE;
		OUTER_ORNG_PLC_DN				:= TRUE;
		AUTO_STP_NO						:= 41;
		END_IF
	
	41: IF NOT ROBO_IN_ORING_ZONE THEN 
		ROBO_GRP_CNTRL.LH_BODY_ROTRY_CMR:= NOT BDY1_PCK_BYPAS;
		ROBO_GRP_CNTRL.RH_BODY_ROTRY_CMR:= NOT BDY2_PCK_BYPAS;
		AUTO_STP_NO						:= 45;
		END_IF
		
	45: IF ROBO_STATUS_FB.BDY_CMR_CHK_POS THEN
		ROBO_GRP_CNTRL.LH_BODY_ROTRY_CMR:= FALSE;
		ROBO_GRP_CNTRL.RH_BODY_ROTRY_CMR:= FALSE;		
		IF NOT BDY1_PCK_BYPAS THEN
		LH_CAMERA_TRIGGER				:= TRUE;
		END_IF
		IF NOT BDY2_PCK_BYPAS THEN
		RH_CAMERA_TRIGGER				:= TRUE;
		END_IF
		AUTO_STP_NO						:= 46;
		END_IF
		ROBO_GRP_CNTRL.LH_BODY_ROTRY_CMR:= FALSE;
		ROBO_GRP_CNTRL.RH_BODY_ROTRY_CMR:= FALSE;
		CMR_TMR(IN:=(AUTO_STP_NO=45), PT:= T#500MS, Q=> , ET=> );
		IF CMR_TMR.Q THEN
		AUTO_STP_NO						:= 46;	
		END_IF
			
	
	46: IF CMR_RESULT_DN THEN
		AUTO_STP_NO						:= 47;
		O_RNG_CHK_DN					:= TRUE;
		END_IF
		PROCESS_DONE					:= FALSE;

	47: ROBO_GRP_CNTRL.LH_BODY_ROTRY_WRK:= NOT BDY1_PCK_BYPAS;
		ROBO_GRP_CNTRL.RH_BODY_ROTRY_WRK:= NOT BDY2_PCK_BYPAS;
		IF (ROBO_GRP_STUS.LH_BDY_ROTRY_WRK_FB OR BDY1_PCK_BYPAS) AND (ROBO_GRP_STUS.RH_BDY_ROTRY_WRK_FB OR BDY2_PCK_BYPAS) THEN
		AUTO_STP_NO						:= 50;
		END_IF
		
	50: IF LH_CMR_ORNG_OK AND RH_CMR_ORING_OK THEN
		ROBO_GRP_CNTRL.LH_BODY_ROTRY_WRK:= FALSE;
		ROBO_GRP_CNTRL.RH_BODY_ROTRY_WRK:= FALSE;
		IF STN_ENABLE THEN
		ROBO_CTRL_WRD.BDY_ORNG_PLC_POS	:= TRUE;
		ROBO_CTRL_WRD.BDY_CMR_CHK_POS	:= TRUE;
		ROBO_CTRL_WRD.BDY_MVE_PLC_POS	:= TRUE;
		AUTO_STP_NO						:= 55;			
		END_IF	
		ELSIF NOT LH_CMR_ORNG_OK AND NOT RH_CMR_ORING_OK THEN
		ROBO_CTRL_WRD.ROBO_REJ_POS		:= TRUE;
		AUTO_STP_NO						:= 200;
		ELSIF (NOT LH_CMR_ORNG_OK AND RH_CMR_ORING_OK) OR (LH_CMR_ORNG_OK AND NOT RH_CMR_ORING_OK) THEN
		IF STN_ENABLE THEN
		ROBO_CTRL_WRD.BDY_ORNG_PLC_POS	:= TRUE;
		ROBO_CTRL_WRD.BDY_CMR_CHK_POS	:= TRUE;
		ROBO_CTRL_WRD.BDY_MVE_PLC_POS	:= TRUE;
		AUTO_STP_NO						:= 300;	
		END_IF			
		END_IF
		
	55: IF ROBO_STATUS_FB.BDY_MVE_PLC_POS THEN
		IF NOT BDY1_PCK_BYPAS AND NOT BDY2_PCK_BYPAS THEN
		ROBO_GRP_CNTRL.LH_BODY_GRIP_HOM	:= TRUE;
		ROBO_GRP_CNTRL.RH_BODY_GRIP_HME	:= TRUE;
		END_IF
		IF BDY1_PCK_BYPAS AND NOT BDY2_PCK_BYPAS THEN
		ROBO_GRP_CNTRL.RH_BODY_GRIP_HME	:= TRUE;
		END_IF
		IF NOT BDY1_PCK_BYPAS AND BDY2_PCK_BYPAS THEN
		ROBO_GRP_CNTRL.LH_BODY_GRIP_HOM	:= TRUE;
		END_IF
		IF (ROBO_GRP_STUS.LH_BDY_GRP_HOM_FB OR BDY1_PCK_BYPAS) AND (ROBO_GRP_STUS.RH_BDY_GRP_HME_FB OR BDY2_PCK_BYPAS) THEN
		OP10_CURR_MOVER					:= OP10_STN_MOVER;
		IF (OP10_CURR_MOVER=OP10_STN_MOVER)	THEN
		AUTO_STP_NO						:= 60;	
		END_IF			
		END_IF
		END_IF
		
	60: F_TRE_ANGLE_CHK_DN				:= FALSE;
		OUTER_ORNG_PLC_DN				:= FALSE;
		O_RNG_CHK_DN					:= FALSE;
		ROBO_GRP_CNTRL.LH_BODY_GRIP_HOM	:= FALSE;
		ROBO_GRP_CNTRL.RH_BODY_GRIP_HME	:= FALSE;			
		ROBO_CTRL_WRD.BDY_S_PCK_POSITION:= TRUE;
		ROBO_CTRL_WRD.BDY_ORNG_PLC_POS	:= FALSE;
		ROBO_CTRL_WRD.BDY_MVE_PLC_POS	:= FALSE;
		ROBO_CTRL_WRD.BDY_CMR_CHK_POS	:= FALSE;
		LH_PART_STATUS					:=	10;
		IF (ROBO_GRP_STUS.LH_BDY_GRP_HOM_FB AND NOT BDY1_PCK_BYPAS) THEN
		LH_PART_STATUS					:=	10;
		ELSIF (*(ROBO_GRP_STUS.LH_BDY_GRP_HOM_FB AND*)BDY1_PCK_BYPAS THEN
		LH_PART_STATUS					:=	10;	
		END_IF	
		IF (ROBO_GRP_STUS.RH_BDY_GRP_HME_FB AND NOT BDY2_PCK_BYPAS) THEN
		RH_PART_STATUS					:=	10;
		ELSIF (*(ROBO_GRP_STUS.RH_BDY_GRP_HME_FB AND*)BDY2_PCK_BYPAS THEN	
		RH_PART_STATUS					:=	10;			
		END_IF
		IF (LH_PART_STATUS=10 OR LH_PART_STATUS=11) AND (RH_PART_STATUS=10 OR RH_PART_STATUS=11) THEN
		AUTO_STP_NO						:= 65;			
		END_IF
		
	65: IF ROBO_STATUS_FB.ROBO_SAFE_POS THEN
		ROBO_GRP_CNTRL.LH_BODY_ROTRY_HOM:= TRUE;
		ROBO_GRP_CNTRL.RH_BODY_ROTRY_HME:= TRUE;		
		ROBO_CTRL_WRD.BDY_S_PCK_POSITION:= FALSE;
		PROCESS_DONE					:= TRUE;
		//IF GRIPPER_HOME OR TEMP_3 THEN						NEED TO BE CHECKED
		ROBO_GRP_CNTRL.LH_BODY_ROTRY_HOM:= FALSE;
		ROBO_GRP_CNTRL.RH_BODY_ROTRY_HME:= FALSE;
		IF NOT CMP_GRIPPED THEN
		AUTO_STP_NO						:= 0;
		END_IF
		//END_IF
		END_IF
	
	200:IF ROBO_STATUS_FB.ROBO_REJ_POS THEN
		IF BDY1_PCK_BYPAS AND NOT BDY2_PCK_BYPAS THEN
		ROBO_GRP_CNTRL.RH_BODY_GRIP_HME	:= TRUE;
		END_IF
		IF NOT BDY1_PCK_BYPAS AND BDY2_PCK_BYPAS THEN
		ROBO_GRP_CNTRL.LH_BODY_GRIP_HOM	:= TRUE;
		END_IF
		AUTO_STP_NO						:= 60;
		END_IF
		
	300:IF ROBO_STATUS_FB.BDY_MVE_PLC_POS THEN
		IF LH_CMR_ORNG_OK AND NOT RH_CMR_ORING_OK  THEN
		LH_PART_STATUS					:=	10;
		RH_PART_STATUS					:=	10;	
		ROBO_GRP_CNTRL.LH_BODY_GRIP_HOM	:= TRUE;
		END_IF
		IF NOT LH_CMR_ORNG_OK AND RH_CMR_ORING_OK THEN
		LH_PART_STATUS					:=	10;
		RH_PART_STATUS					:=	10;		
		ROBO_GRP_CNTRL.RH_BODY_GRIP_HME	:= TRUE;
		END_IF
		IF (LH_PART_STATUS=10 OR LH_PART_STATUS=11) AND (RH_PART_STATUS=10 OR RH_PART_STATUS=11) THEN
		AUTO_STP_NO						:= 305;				
		END_IF		
		END_IF
	
	305:ROBO_CTRL_WRD.ROBO_REJ_POS		:= TRUE;
		AUTO_STP_NO						:= 310;

	310:IF ROBO_STATUS_FB.ROBO_REJ_POS THEN
		IF LH_CMR_ORNG_OK AND NOT RH_CMR_ORING_OK  THEN
		ROBO_GRP_CNTRL.RH_BODY_GRIP_HME	:= TRUE;
		END_IF
		IF NOT LH_CMR_ORNG_OK AND RH_CMR_ORING_OK THEN
		ROBO_GRP_CNTRL.LH_BODY_GRIP_HOM	:= TRUE;
		END_IF
		IF (LH_PART_STATUS=10 OR LH_PART_STATUS=11) AND (RH_PART_STATUS=10 OR RH_PART_STATUS=11) THEN
		ROBO_CTRL_WRD.BDY_S_PCK_POSITION:= TRUE;
		AUTO_STP_NO						:= 315;				
		END_IF		
		END_IF

	315:IF ROBO_STATUS_FB.ROBO_SAFE_POS THEN
		ROBO_CTRL_WRD.BDY_S_PCK_POSITION:= FALSE;
		AUTO_STP_NO						:= 0;		
		END_IF 
	
END_CASE
END_IF
ELSE
	AUTO_STP_NO							:= 0;
	ROBO_CTRL_WRD.BDY_PCK_POSITION		:= FALSE;
	ROBO_CTRL_WRD.BDY_CMR_CHK_POS		:= FALSE;
	ROBO_CTRL_WRD.BDY_MVE_PLC_POS		:= FALSE;
	ROBO_CTRL_WRD.BDY_S_ORNG_POS		:= FALSE;
	ROBO_CTRL_WRD.BDY_ORNG_PLC_POS		:= FALSE;
	ROBO_CTRL_WRD.ROBO_SAFE_POS			:= FALSE;
	ROBO_GRP_CNTRL.LH_BODY_GRIP_WRK		:= FALSE;
	ROBO_GRP_CNTRL.LH_BODY_GRIP_HOM	    := FALSE;
	ROBO_GRP_CNTRL.RH_BODY_GRIP_WRK	    := FALSE;
	ROBO_GRP_CNTRL.RH_BODY_GRIP_HME	    := FALSE;
	ROBO_GRP_CNTRL.LH_BODY_ROTRY_WRK	:= FALSE;
	ROBO_GRP_CNTRL.LH_BODY_ROTRY_HOM	:= FALSE;
	ROBO_GRP_CNTRL.RH_BODY_ROTRY_WRK	:= FALSE;
	ROBO_GRP_CNTRL.RH_BODY_ROTRY_HME	:= FALSE;
	ROBO_GRP_CNTRL.LH_BODY_RTRY_FITEE	:= FALSE;
	ROBO_GRP_CNTRL.RH_BODY_RTRY_FITEE	:= FALSE;	
	ROBO_GRP_CNTRL.LH_BODY_ROTRY_CMR	:= FALSE;
	ROBO_GRP_CNTRL.RH_BODY_ROTRY_CMR	:= FALSE;	
	PLC_OUTR_ORNG						:= FALSE;
	LH_CAMERA_TRIGGER					:= FALSE;
	RH_CAMERA_TRIGGER					:= FALSE;
(*	CMP_GRIPPED							:= FALSE;
	F_TRE_ANGLE_CHK_DN                  := FALSE;
	OUTER_ORNG_PLC_DN                   := FALSE;
	O_RNG_CHK_DN                        := FALSE;*)
END_IF	

IF START_HOMING THEN
	F_TRE_ANGLE_CHK_DN                  := FALSE;
	OUTER_ORNG_PLC_DN                   := FALSE;
	O_RNG_CHK_DN                        := FALSE;
END_IF


GRIPPER_HOME							:= (ROBO_GRP_STUS.LH_BDY_GRP_HOM_FB OR CMP_GRIPPED OR BDY1_PCK_BYPAS)AND (ROBO_GRP_STUS.RH_BDY_GRP_HME_FB OR CMP_GRIPPED OR BDY2_PCK_BYPAS)AND 
											((ROBO_GRP_STUS.LH_BDY_ROTRY_HOM_FB OR ROBO_GRP_STUS.LH_BDY_ROTRY_ZERO_FB) OR F_TRE_ANGLE_CHK_DN OR BDY1_PCK_BYPAS) AND 
											((ROBO_GRP_STUS.RH_BDY_ROTRY_HME_FB OR ROBO_GRP_STUS.RH_BDY_ROTRY_ZERO_FB) OR F_TRE_ANGLE_CHK_DN OR BDY2_PCK_BYPAS);



IF START_HOMING THEN
	IF ROBO_GRP_OPN THEN
		IF LH_GRP_HME_REF THEN
		ROBO_GRP_CNTRL.LH_BODY_GRIP_HOMING_1:= FALSE;	
		ROBO_GRP_CNTRL.LH_BODY_GRIP_HOM	    := ROBO_GRP_OPN;//NOT(ROBO_GRP_STUS.LH_BDY_GRP_HOM_FB OR CMP_GRIPPED OR BDY1_PCK_BYPAS);		
		ELSE
		ROBO_GRP_CNTRL.LH_BODY_GRIP_HOMING_1:= TRUE;
		LH_GRP_REF(CLK:= LH_BODY_GRIP_HME_DN, Q=> );
		IF LH_GRP_REF.Q THEN
		LH_GRP_HME_REF						:= TRUE;
		ROBO_GRP_CNTRL.LH_BODY_GRIP_HOMING_1:= FALSE;
		END_IF	
		END_IF
		
		IF RH_GRP_HME_REF THEN
		ROBO_GRP_CNTRL.RH_BODY_GRIP_HOMING_1:=FALSE;
		ROBO_GRP_CNTRL.RH_BODY_GRIP_HME	    :=ROBO_GRP_OPN;// NOT(ROBO_GRP_STUS.RH_BDY_GRP_HME_FB OR CMP_GRIPPED OR BDY2_PCK_BYPAS);		
		ELSE
		ROBO_GRP_CNTRL.RH_BODY_GRIP_HOMING_1:=TRUE;
		RH_GRP_REF(CLK:= RH_BODY_GRIP_HME_DN, Q=> );	
		IF RH_GRP_REF.Q THEN
		RH_GRP_HME_REF						:= TRUE;
		ROBO_GRP_CNTRL.RH_BODY_GRIP_HOMING_1:=FALSE;	
		END_IF	
		END_IF
	END_IF
	
	IF ROBO_IN_HOME THEN
	IF LH_ROTRY_HME_REF THEN
	ROBO_GRP_CNTRL.LH_BODY_ROTRY_HOMING_1:= FALSE;	
	ROBO_GRP_CNTRL.LH_BODY_ROTRY_HOM	:= NOT((ROBO_GRP_STUS.LH_BDY_ROTRY_HOM_FB OR ROBO_GRP_STUS.LH_BDY_ROTRY_ZERO_FB) OR F_TRE_ANGLE_CHK_DN OR BDY1_PCK_BYPAS);	
	ELSE
	ROBO_GRP_CNTRL.LH_BODY_ROTRY_HOMING_1:= TRUE;
	LH_ROTRY_REF(CLK:= LH_BODY_ROTRY_HME_DN, Q=> );
	IF LH_ROTRY_REF.Q THEN
	LH_ROTRY_HME_REF					 := TRUE;
	ROBO_GRP_CNTRL.LH_BODY_ROTRY_HOMING_1:= FALSE;	
	END_IF
	END_IF
	
	IF RH_ROTRY_HME_REF THEN
	ROBO_GRP_CNTRL.RH_BODY_ROTRY_HOMING_1:= FALSE;
	ROBO_GRP_CNTRL.RH_BODY_ROTRY_HME	:= NOT((ROBO_GRP_STUS.RH_BDY_ROTRY_HME_FB OR ROBO_GRP_STUS.RH_BDY_ROTRY_ZERO_FB) OR F_TRE_ANGLE_CHK_DN OR BDY2_PCK_BYPAS);	
	ELSE
	ROBO_GRP_CNTRL.RH_BODY_ROTRY_HOMING_1:= TRUE;
	RH_ROTRY_REF(CLK:= RH_BODY_ROTRY_HME_DN, Q=> );
	IF RH_ROTRY_REF.Q THEN
	RH_ROTRY_HME_REF					 := TRUE;
	ROBO_GRP_CNTRL.RH_BODY_ROTRY_HOMING_1:= FALSE;	
	END_IF
	END_IF	
	END_IF	
END_IF

END_FUNCTION_BLOCK

// ---- FB/Axis/FB_Axis.TcPOU
FUNCTION_BLOCK FB_Axis
VAR_INPUT
	bAxis1_Ref_Switch 	 : BOOL;//HW-IN
	bInit 				 : BOOL;
	bErrorReset			 : BOOL;//FP Reset Axis Error
	bEnable 			 : BOOL;//Power on
	bMoveVelocity 		 : BOOL;
	bHalt				 : BOOL;//Stop Absolute or Relative movement
	bManualMode			 : BOOL;
	fHomePos 			 : LREAL := 0.0;
	fOverride 			 : LREAL := 100.0;
	fTargetPosition 	 : LREAL ;//:=  10.0;
	fTargetVelocity 	 : LREAL ; //:= 100.0;
	fAcc				 : LREAL; //:= 100.0;
	fDec				 : LREAL; //:= 100.0;
	Servo_High_Limit	 : LREAL;
	Servo_Low_Limit	 	 : LREAL;
	WARNING_LIMIT		 : LREAL;
	LIMIT_BYPASS		 : BOOL;	
	Safe_move_Conditions : BOOL;
	HME_WRITE_ADD		 : UDINT;
	Torque_limit_perent	 : REAL;
END_VAR
VAR_IN_OUT
	Axis 				: AXIS_REF;
	bHome 				: BOOL;
	bSetPosition		: BOOL;//Set Position to HomePos
	bMoveAbsolute 		: BOOL;
	bMoveRelative 		: BOOL;
	bMoveTorque			: BOOL;
    stManualModeAxis  	: stManualModeAxis;
	bmove_home			: BOOL;
END_VAR

VAR_OUTPUT
	sAxisState			: STRING := '';
	bAxis_ready			: BOOL := 0;
	bAxisInPosition		: BOOL := 0;//In Position or In Target Velocity
	bAxisError			: BOOL := 0;
	bAxisEnabled 		: BOOL := 0;//Power ON
	bAxisHomed			: BOOL := 0;
	bSetPositionDone	: BOOL := 0;
	bHaltDone			: BOOL := 0;
	bSTOPDone			: BOOL := 0;
	bHomeDone			: BOOL := 0;
	bDone				: BOOL := 0;//bMoveAbsolute + bMoveRelative
	bTorqueReached		: BOOL := 0;
	bsafe_to_move		: BOOL;
	baxis_in_home_pos	: BOOL;
	bABS_Pos_done		: BOOL;
	Actual_position		: LREAL;
	Actual_velocity		: LREAL;
	Actual_Torque		: LREAL;
    SERVO_LIMIT_WARNING	: BOOL;
	TORQUE_LIMIT		: UINT; 
	POS_TORQUE_LIMIT 	: UINT;
	NEG_TORQUE_LIMIT	: UINT;	
	
	
END_VAR
VAR
	temp : LREAL;
	fbAxisReset					: MC_Reset;
	fbAxisPower					: MC_Power;
	fbAxisStop        			: MC_Stop;
	fbAxisHalt        			: MC_Halt;
	fbAxisHome					: MC_Home;
	fbAxisSetPosition 			: MC_SetPosition;
	fbAxisJog 					: MC_Jog;
	fbAxisMoveAbsolute			: MC_MoveAbsolute;
	fbAxisMoveRelative 			: MC_MoveRelative;
	fbAxisMoveVelocity			: MC_MoveVelocity;
	fbAxisTorqueControl			: MC_TorqueControl;
//Brake Controll
	fbEcCoeSdoRead				: FB_EcCoeSdoRead;
	fbEcCoeSdoWrite				: FB_EcCoeSdoWrite;
	mcReadDriveAddress 			: MC_ReadDriveAddress;
    vendorId   					: BOOL;//Struct HMI Brake open
	bBrakeStateOld 				: BOOL;

//Status Information
	bAxisIsEnabled 				: BOOL;
	bAxisIsHomed 				: BOOL;
	bAxisInError 				: BOOL;
	fActualTorque 				: LREAL;	

//Allgemein
	iSchritt 					: ENUM_Axis;
	bHMFPErrorReset 			: BOOL;
	bFPErrorReset 				: BOOL;
	
	bAxisResetExecute			: BOOL;
	bAxisPowerExecute			: BOOL;
	bAxisStopExecute        	: BOOL;
	bAxisHaltExecute        	: BOOL;
	bAxisHomeExecute			: BOOL;
	bAxisSetPositionExecute 	: BOOL;
	bAxisMoveAbsoluteExecute	: BOOL;
	bAxisMoveRelativeExecute 	: BOOL;
	bAxisMoveVelocityExecute	: BOOL;
	bAxisJogExecutePos 			: BOOL;
	bAxisJogExecuteNeg 			: BOOL;
	bAxisMoveTorqueExecute		: BOOL;
	fHMTargetPosition			: LREAL;
	fHMTargetVelocity			: LREAL;
	
	bFPManualReset				: BOOL;
	bHMFPManualReset			: BOOL;
	
	homeMode					: MC_HomingMode;
	FB_SoEReset					: FB_SoEReset;
	bHardwareReset				: BOOL;

	st_Trq_options 				: St_TorqueControlOptions;
	//temp						: BOOL;
	moving_home					: INT;
	bABS_done					: BOOL;
	busy: BOOL;
	act: BOOL;
	id: UDINT;
///////////////////////////////////////////////////////////////////////////////////////////////////	
	FB_GetLocalAmsNetId_system		: FB_GetLocalAmsNetId;
	ADSREAD_set_val					: ADSREAD;
	ADSWRITE_Set_Val				: ADSWRITE;
	bSet_Encoder_Zero_Rtrig			: R_trig;
	F_TRIG1							: F_TRIG;
	tDummy							: Ton;
	lrRead_set_Value				: LREAL;
	Step							: INT;
	bSet_Encoder_Zero				: BOOL;
	bRead_set_Value					: BOOL;
	bWrite_set_Value				: BOOL;
	bHome_ref_done					: BOOL;
	TRIAL							: BOOL;
	home_pressed					: BOOL;
//	stAxis:AXIS_REF;
//	MC_Power1: MC_Power;
//	bEnable: BOOL;


	LEG_LIMIT: BOOL;
	POS_LIMIT: BOOL;
	AUTO_TARGET_POSITION: LREAL;
	MANUAL_TARGET_POSITION: LREAL;
	START_TIMER: TON;
END_VAR
VAR_TEMP
 	//tmpVelocityDirection		: MC_Direction;
	tmpStManualModeAxis	  		: stManualModeAxis;
	btmpFPBrake					: BOOL;
//	tmpVelocityDirection        : MC_Direction;
END_VAR


VAR PERSISTENT
	aa					: DINT;
	lrWrite_set_Value	: LREAL;
	HOMING_VALUE		: LREAL;
END_VAR

//Init
bHaltDone := FALSE;
bSTOPDone := FALSE;

//Read Axis Status	
	bAxisIsEnabled := axis.NcToPlc.StateDWord.0;
	bAxisIsHomed := axis.NcToPlc.StateDWord.1 OR TRIAL;
	bAxisInError := axis.NcToPlc.StateDWord.31;
	fActualTorque := axis.NcToPlc.ActTorque;
    Axis.ReadStatus(); // PHU: fill its own status bits.
//FP Error Reset
	bFPErrorReset := bErrorReset AND NOT bHMFPErrorReset;
	bHMFPErrorReset := bErrorReset;
	
	bFPManualReset:= stManualModeAxis.reset AND NOT bHMFPManualReset;
	bHMFPManualReset:= stManualModeAxis.reset;
	
// Manual Mode
IF bManualMode THEN
	
	stManualModeAxis.stationModeAutoManual:= FALSE;	
	IF 	stManualModeAxis.jogPos THEN
		tmpStManualModeAxis.jogPos := TRUE;
	ELSE
		tmpStManualModeAxis.jogPos := FALSE;		
	END_IF
	IF 	stManualModeAxis.jogNeg THEN
		tmpStManualModeAxis.jogNeg := TRUE;
	ELSE
		tmpStManualModeAxis.jogNeg := FALSE;		
	END_IF
		
ELSE
	stManualModeAxis.jogPos := FALSE;
	stManualModeAxis.jogNeg := FALSE;
	stManualModeAxis.reset := FALSE;
	StManualModeAxis.openBrake:= FALSE;
	stManualModeAxis.homing:= FALSE;
	stManualModeAxis.moveAbsolute:= FALSE;
	stManualModeAxis.moveRelative:= FALSE;
	stManualModeAxis.moveVelocity:= FALSE;
	
	tmpStManualModeAxis.jogPos := FALSE;		
	tmpStManualModeAxis.jogNeg := FALSE;	
	
	
	
	stManualModeAxis.stationModeAutoManual:= TRUE;

END_IF


//###################################################################################
//###################################################################################	
	
//###################################################################################
//###################################################################################

	CASE iSchritt OF 
		
	ENUM_Axis.Init 			://init all MC
								bAxisResetExecute				:= FALSE;
								bAxisPowerExecute				:= FALSE;
								bAxisStopExecute        		:= FALSE;
								bAxisHaltExecute        		:= FALSE;
								bAxisHomeExecute				:= FALSE;
								bAxisSetPositionExecute 		:= FALSE;
								bAxisJogExecutePos 				:= FALSE;
								bAxisJogExecuteNeg 				:= FALSE;
								bAxisMoveAbsoluteExecute		:= FALSE;
								bAxisMoveRelativeExecute 		:= FALSE;
								bAxisMoveVelocityExecute		:= FALSE;
								
								iSchritt := ENUM_Axis.PowerOFF;
								

	ENUM_Axis.PowerOFF		: 	//Power off
								bAxisPowerExecute		:= FALSE;
								IF bInit THEN
									iSchritt := ENUM_Axis.Init;
								ELSIF bAxisInError THEN
									iSchritt := ENUM_Axis.Error;
								ELSIF bEnable  THEN
									iSchritt := ENUM_Axis.PowerON;
								END_IF
								
	ENUM_Axis.Error			:	//Error
								bAxisPowerExecute			  := FALSE;
								bMoveAbsolute				  := FALSE;
								bMoveRelative			   	  := FALSE;
								stManualModeAxis.moveAbsolute := FALSE;
								stManualModeAxis.moveRelative := FALSE;
								IF bInit THEN
									iSchritt := ENUM_Axis.Init;
								ELSIF bFPErrorReset OR bFPManualReset THEN
									iSchritt := ENUM_Axis.Reset;
								END_IF
	ENUM_Axis.Reset			: //Error Reset
								IF NOT fbAxisReset.Busy THEN
									bAxisResetExecute 		:= TRUE;
									bHardwareReset			:= axis.NcToPlc.StateDWord.28;
								END_IF;
								IF bInit THEN
									bAxisResetExecute 		:= FALSE;
									iSchritt := ENUM_Axis.Init;
								ELSIF fbAxisReset.Error (*OR bAxisInError *)THEN
									bAxisResetExecute 	:= FALSE;
									iSchritt := ENUM_Axis.Error;
								ELSIF fbAxisReset.Done AND NOT bAxisInError THEN
									bAxisResetExecute 	:= FALSE;
									IF  bAxisInError THEN
										iSchritt := ENUM_Axis.Error;
									ELSE
										iSchritt := ENUM_Axis.PowerOFF;
									END_IF
								END_IF

	ENUM_Axis.PowerON		:	//Enable - Power on
								bAxisPowerExecute := TRUE;
								IF bInit THEN
									bAxisPowerExecute 	:= FALSE;
									iSchritt := ENUM_Axis.Init;
								ELSIF NOT benable THEN
									iSchritt:= enum_axis.PowerOFF;
								ELSIF fbAxisPower.Error OR bAxisInError THEN
									bAxisPowerExecute 	:= FALSE;
									iSchritt := ENUM_Axis.Error;
								ELSIF fbAxisPower.Status THEN
									iSchritt := ENUM_Axis.Ready;
								END_IF
	ENUM_Axis.Stop			://Axis Stop
								bAxisStopExecute := TRUE;
								IF bInit THEN
									bAxisStopExecute 	:= FALSE;
									iSchritt := ENUM_Axis.Init;
								ELSIF NOT benable THEN
									bAxisStopExecute 	:= FALSE;
									iSchritt:= enum_axis.PowerOFF;	
								ELSIF fbAxisStop.Error OR bAxisInError THEN
									bAxisStopExecute := FALSE;
									iSchritt := ENUM_Axis.Error;
								ELSIF fbAxisStop.Done THEN
									bSTOPDone	:= TRUE;
									bAxisStopExecute 	:= FALSE;
									iSchritt := ENUM_Axis.PowerOFF;
								END_IF
	ENUM_Axis.Halt			://Axis Halt
								bAxisHaltExecute := TRUE;
								IF bInit THEN
									bAxisHaltExecute 	:= FALSE;
									iSchritt := ENUM_Axis.Init;
								ELSIF NOT benable THEN
									bAxisHaltExecute 	:= FALSE;
									iSchritt:= enum_axis.PowerOFF;	
								ELSIF bAxisInError THEN
									bAxisHaltExecute := FALSE;
									iSchritt := ENUM_Axis.Error;
								ELSIF fbAxisHalt.Error (*OR bAxisInError *)THEN
									bAxisHaltExecute := FALSE;
									iSchritt := ENUM_Axis.Stop;
								ELSIF fbAxisHalt.Done THEN
									bHaltDone := TRUE;
									bAxisHaltExecute := FALSE;
									iSchritt := ENUM_Axis.Ready;
								END_IF
	ENUM_Axis.Ready			: 	//Wait for command
								bAxisInPosition := FALSE;
								bHomeDone := FALSE;
								bSetPositionDone := FALSE;
								IF bInit THEN
									iSchritt := ENUM_Axis.Init;
								ELSIF NOT benable THEN
									iSchritt:= enum_axis.PowerOFF;		
								ELSIF bAxisInError THEN
									iSchritt := ENUM_Axis.Error;
								ELSE
									IF bHome OR stManualModeAxis.homing THEN
										//iSchritt := ENUM_Axis.Homing;
										home_pressed:=bHome;
										home_pressed:=TRUE;
									ELSIF bSetPosition THEN
										//	iSchritt := ENUM_Axis.SetPosition;
										home_pressed:=bSetPosition;
										home_pressed:=TRUE;
									ELSIF bAxisIsHomed THEN
										IF tmpStManualModeAxis.jogPos THEN
											iSchritt := ENUM_Axis.JogPos;
										ELSIF tmpStManualModeAxis.jogNeg THEN
											iSchritt := ENUM_Axis.JogNeg;
										ELSIF bMoveAbsolute OR stManualModeAxis.moveAbsolute  THEN
											iSchritt := ENUM_Axis.MoveAbsolute;
										ELSIF bMoveRelative OR stManualModeAxis.moveRelative THEN
											iSchritt := ENUM_Axis.MoveRelative;
										ELSIF bMoveVelocity OR stManualModeAxis.moveVelocity THEN
											iSchritt := ENUM_Axis.MoveVelocity;
										ELSIF bMoveTorque OR stManualModeAxis.moveTorque THEN
											iSchritt := ENUM_Axis.MoveTorque;
										END_IF
									END_IF	
								END_IF							
	ENUM_Axis.Homing		://Homing
								IF NOT fbAxisHome.Busy THEN
									bAxisHomeExecute := TRUE;
								END_IF;
								IF bInit THEN
									bAxisHomeExecute 	:= FALSE;
									iSchritt := ENUM_Axis.Init;
								ELSIF NOT benable THEN
									bAxisHomeExecute:= FALSE;
									iSchritt:= enum_axis.PowerOFF;	
								ELSIF fbAxisHome.Error OR bAxisInError THEN
									bAxisHomeExecute:= FALSE;
									iSchritt := ENUM_Axis.Error;
								ELSIF fbAxisHome.Done THEN
									bHomeDone := TRUE;
									bHome := FALSE;
									stManualModeAxis.homing:= FALSE;
									bAxisHomeExecute:= FALSE;
									iSchritt := ENUM_Axis.Ready;
								END_IF
	
	ENUM_Axis.SetPosition	://Enable - Power on
								IF NOT fbAxisSetPosition.Busy THEN
									bAxisSetPositionExecute := TRUE;
								END_IF;
								IF bInit THEN
									bAxisSetPositionExecute 	:= FALSE;
									iSchritt := ENUM_Axis.Init;
								ELSIF NOT benable THEN
									bAxisSetPositionExecute 	:= FALSE;
									iSchritt:= enum_axis.PowerOFF;		
								ELSIF fbAxisSetPosition.Error OR bAxisInError THEN
									bAxisSetPositionExecute 	:= FALSE;
									iSchritt := ENUM_Axis.Error;
								ELSIF fbAxisSetPosition.Done THEN
									bAxisSetPositionExecute 	:= FALSE;
									bSetPositionDone := TRUE;
									bSetPosition := FALSE;
									iSchritt := ENUM_Axis.Ready;
								END_IF

	ENUM_Axis.JogPos		://Jog positive direction
								IF NOT fbAxisJog.Busy THEN
									bAxisJogExecutePos 		:= TRUE;
								END_IF;
								
								IF bInit THEN
									bAxisJogExecutePos 	:= FALSE;
									iSchritt := ENUM_Axis.Init;
								ELSIF NOT benable THEN
									bAxisJogExecutePos 	:= FALSE;
									iSchritt:= enum_axis.PowerOFF;			
								ELSIF fbAxisJog.Error OR bAxisInError THEN
									bAxisJogExecutePos 		:= FALSE;
									iSchritt := ENUM_Axis.Error;
								ELSIF NOT tmpStManualModeAxis.jogPos THEN
									bAxisJogExecutePos 		:= FALSE;
									iSchritt := ENUM_Axis.Ready;
								END_IF;
	ENUM_Axis.JogNeg		://Jog negative direction
								IF NOT fbAxisJog.Busy THEN
									bAxisJogExecuteNeg 		:= TRUE;
								END_IF;
								
								IF bInit THEN
									bAxisJogExecuteNeg 	:= FALSE;
									iSchritt := ENUM_Axis.Init;
								ELSIF NOT benable THEN
									bAxisJogExecuteNeg 	:= FALSE;
									iSchritt:= enum_axis.PowerOFF;		
								ELSIF fbAxisJog.Error OR bAxisInError THEN
									bAxisJogExecuteNeg 		:= FALSE;
									iSchritt := ENUM_Axis.Error;
								ELSIF NOT tmpStManualModeAxis.jogNeg THEN
									bAxisJogExecuteNeg 		:= FALSE;
									iSchritt := ENUM_Axis.Ready;
								END_IF;
	ENUM_Axis.MoveAbsolute	://MoveAbsolute
								IF NOT fbAxisMoveAbsolute.Busy THEN
									bAxisMoveAbsoluteExecute := TRUE;
								END_IF;
								IF bInit THEN
									bAxisMoveAbsoluteExecute 	:= FALSE;
									iSchritt := ENUM_Axis.Init;
								ELSIF NOT benable THEN
									bAxisMoveAbsoluteExecute 	:= FALSE;
									iSchritt:= enum_axis.PowerOFF;		
								ELSIF fbAxisMoveAbsolute.Error OR bAxisInError THEN
									bAxisMoveAbsoluteExecute :=FALSE;
									iSchritt := ENUM_Axis.Error;
								ELSIF bHalt THEN
									bMoveAbsolute :=FALSE;
									stManualModeAxis.moveAbsolute:= FALSE;
									bAxisMoveAbsoluteExecute :=FALSE;
									iSchritt := ENUM_Axis.Halt;
								ELSIF fbAxisMoveAbsolute.Done THEN
								//ELSIF fbAxisMoveAbsolute.Done AND NOT bMoveAbsolute THEN
									bMoveAbsolute :=FALSE;
									stManualModeAxis.moveAbsolute:= FALSE;
									bAxisInPosition := TRUE;
									bAxisMoveAbsoluteExecute :=FALSE;
									iSchritt := ENUM_Axis.Ready;
								END_IF;
	ENUM_Axis.MoveRelative	://MoveRelative
								IF NOT fbAxisMoveRelative.Busy THEN
									bAxisMoveRelativeExecute := TRUE;
								END_IF;
								IF bInit THEN
									bAxisMoveRelativeExecute 	:= FALSE;
									iSchritt := ENUM_Axis.Init;
								ELSIF NOT benable THEN
									bAxisMoveRelativeExecute 	:= FALSE;
									iSchritt:= enum_axis.PowerOFF;		
								ELSIF fbAxisMoveRelative.Error OR bAxisInError THEN
									bAxisMoveRelativeExecute :=FALSE;
									iSchritt := ENUM_Axis.Error;
								ELSIF bHalt THEN
									bMoveRelative :=FALSE;
									stManualModeAxis.moveRelative:= FALSE;
									bAxisMoveRelativeExecute :=FALSE;
									iSchritt := ENUM_Axis.Halt;
								ELSIF fbAxisMoveRelative.Done THEN
									bMoveRelative :=FALSE;
									stManualModeAxis.moveRelative:= FALSE;
									bAxisInPosition := TRUE;
									bAxisMoveRelativeExecute :=FALSE;
									iSchritt := ENUM_Axis.Ready;
								END_IF;
	ENUM_Axis.MoveVelocity	://MoveVelocity
								IF NOT fbAxisMoveVelocity.Busy THEN
									bAxisMoveVelocityExecute := TRUE;				
								END_IF;
								
								bAxisInPosition := fbAxisMoveVelocity.InVelocity;
								IF bInit THEN
									bAxisMoveVelocityExecute 	:= FALSE;
									bAxisInPosition := FALSE;
									iSchritt := ENUM_Axis.Init;
								ELSIF NOT benable THEN
									bAxisMoveVelocityExecute 	:= FALSE;
									iSchritt:= enum_axis.PowerOFF;		
								ELSIF fbAxisMoveVelocity.Error OR bAxisInError THEN
									bAxisInPosition := FALSE;
									bAxisMoveVelocityExecute :=FALSE;
									iSchritt := ENUM_Axis.Error;
								ELSIF NOT bMoveVelocity AND NOT stManualModeAxis.moveVelocity THEN
									bAxisInPosition := FALSE;
									bAxisMoveVelocityExecute :=FALSE;
									iSchritt := ENUM_Axis.Halt;
								END_IF;
								
	ENUM_Axis.MoveTorque  :		IF NOT fbAxisTorqueControl.Busy THEN
									bAxisMoveTorqueExecute := TRUE;
								END_IF;
								IF bInit THEN
									bAxisMoveTorqueExecute 	:= FALSE;
									iSchritt := ENUM_Axis.Init;
								ELSIF NOT benable THEN
									bAxisMoveTorqueExecute 	:= FALSE;
									iSchritt:= enum_axis.PowerOFF;		
								ELSIF fbAxisTorqueControl.Error OR bAxisInError THEN
									bAxisMoveTorqueExecute :=FALSE;
									iSchritt := ENUM_Axis.Error;
								ELSIF bHalt THEN
									bMoveTorque	 :=FALSE;
									stManualModeAxis.moveTorque:= FALSE;
									bAxisMoveTorqueExecute :=FALSE;
									iSchritt := ENUM_Axis.Halt;
								ELSIF fbAxisTorqueControl.InTorque THEN
								//ELSIF fbAxisMoveAbsolute.Done AND NOT bMoveAbsolute THEN
									bMoveTorque :=FALSE;
									stManualModeAxis.moveTorque:= FALSE;
									bAxisInPosition := TRUE;
									bAxisMoveTorqueExecute :=FALSE;
									iSchritt := ENUM_Axis.Ready;
								END_IF;					

	END_CASE;
	
	
	stManualModeAxis.axisState:= TO_STRING(iSchritt);
//###################################################################################
//###################################################################################
//###################################################################################
//###################################################################################



fbAxisReset(
	Axis:= Axis, 
	Execute:= bAxisResetExecute , 
	Done=> , 
	Busy=> , 
	Error=> , 
	ErrorID=> );
	
fbAxisPower(
	Axis:= Axis, 
	Enable:= bAxisPowerExecute AND NOT home_pressed AND TRIAL, 
	Enable_Positive:= bAxisPowerExecute, 
	Enable_Negative:= bAxisPowerExecute, 
	Override:= fOverride, 
	//BufferMode:= , 
	//Options:= , 
	Status=> , 
	Busy=> , 
	Active=> , 
	Error=> , 
	ErrorID=> );
	
fbAxisStop(
	Axis:= Axis, 
	Execute:= bAxisStopExecute, 
	Deceleration:= fDec, 
	Jerk:= 0, 
	//Options:= , 
	Done=> , 
	Busy=> , 
	Active=> , 
	CommandAborted=> , 
	Error=> , 
	ErrorID=> );
	
fbAxisHalt(
	Axis:= Axis, 
	Execute:= bAxisHaltExecute, 
	Deceleration:= fDec, 
	Jerk:= 0, 
	//BufferMode:= , 
	//Options:= , 
	Done=> , 
	Busy=> , 
	Active=>, 
	CommandAborted=> , 
	Error=> , 
	ErrorID=> );

//Homingmode
IF bAxisHomeExecute THEN
	//HomeMode := MC_DefaultHoming;
	HomeMode := MC_Direct;
ELSIF bAxisSetPositionExecute THEN
	//HomeMode := MC_ForceCalibration;
		HomeMode := MC_Direct;
END_IF;


IF bManualMode THEN
	fHMTargetPosition:= MANUAL_TARGET_POSITION;//MANUAL_TARGET_POSITION;
	fHMTargetVelocity:= stManualModeAxis.targetVelocity;
ELSE
	fHMTargetPosition:=AUTO_TARGET_POSITION;
	fHMTargetVelocity:=fTargetVelocity;
END_IF


fbAxisHome(
	Axis:= Axis, 
	Execute:= bAxisHomeExecute OR bAxisSetPositionExecute , 
	Position:= fHomePos, 
	HomingMode:= HomeMode, //MC_DefaultHoming,//, MC_Block
	//BufferMode:= , 
	Options:= , 
	bCalibrationCam:= bAxis1_Ref_Switch, 
	Done=> , 
	Busy=> , 
	Active=> , 
	CommandAborted=> , 
	Error=> , 
	ErrorID=> );

fbAxisSetPosition(
	Axis:= Axis, 
	Execute:= bAxisSetPositionExecute, 
	Position:= fHomePos, 
	Mode:= FALSE, (* RELATIVE=True, ABSOLUTE=False (Default) *)
	//Options:= , 
	Done=> , 
	Busy=> , 
	Error=> , 
	ErrorID=> );

fbAxisJog(
	Axis:= Axis, 
	JogForward:=bAxisJogExecutePos AND (POS_LIMIT OR LIMIT_BYPASS),
	JogBackwards:= bAxisJogExecuteNeg AND (LEG_LIMIT OR LIMIT_BYPASS),
	//Mode:= MC_JOGMODE_STANDARD_SLOW, //MC_JOGMODE_STANDARD_SLOW, //MC_JOGMODE_STANDARD_FAST, //MC_JOGMODE_CONTINOUS, //MC_JOGMODE_INCHING, //MC_JOGMODE_INCHING_MODULO
	//Position:= 0, 
	Velocity:= stManualModeAxis.targetVelocity, 
	Acceleration:= fAcc, 
	Deceleration:= fDec, 
	Jerk:= 0, 
	Done=> , 
	Busy=> , 
	Active=> , 
	CommandAborted=> , 
	Error=> , 
	ErrorID=> );
	
fbAxisMoveAbsolute(
	Axis:= Axis, 
	Execute:= bAxisMoveAbsoluteExecute, 
	Position:= fHMTargetPosition,
	Velocity:= ABS(fHMTargetVelocity),
	Acceleration:= fAcc,
	Deceleration:= fDec,
	Jerk:= 0, 
	//BufferMode:= , 
	//Options:= , 
	Done=> , 
	Busy=> , 
	Active=> (bABS_done) , 
	CommandAborted=> , 
	Error=> , 
	ErrorID=> );

bABS_Pos_done:=NOT (bABS_done);//fbAxisMoveAbsolute.Done;
	
fbAxisMoveRelative(
	Axis:= Axis, 
	Execute:= bAxisMoveRelativeExecute, 
	Distance:= fHMTargetPosition, 
	Velocity:= fHMTargetVelocity, 
	Acceleration:= fAcc, 
	Deceleration:= fDec, 
	Jerk:= 0, 
	//BufferMode:= , 
	//Options:= , 
	Done=> , 
	Busy=> , 
	Active=> , 
	CommandAborted=> , 
	Error=> , 
	ErrorID=> );

IF 	fHMTargetVelocity >= 0 THEN  // fHMTargetVelocity>= 0
	fbAxisMoveVelocity.Direction:= MC_Positive_Direction;
ELSE
	fbAxisMoveVelocity.Direction:= MC_Negative_Direction;
END_IF
	
fbAxisMoveVelocity(
	Axis:= Axis, 
	Execute:= bAxisMoveVelocityExecute, 
	Velocity:=ABS(fHMTargetVelocity), 
	Acceleration:= fAcc, 
	Deceleration:= fDec, 
	Jerk:= 0, 
	Direction:= ,//MC_Negative_Direction ,//OR MC_Positive_Direction, //tmpVelocityDirection,//MC_Undefined_Direction, //MC_Shortest_Way, //MC_Positive_Direction, //MC_Negative_Direction,
	//BufferMode:= , 
	//Options:= , 
	InVelocity=> , 
	Busy=> , 
	Active=> , 
	CommandAborted=> , 
	Error=> , 
	ErrorID=> );
	
//Brake controll
vendorId	:= StManualModeAxis.openBrake;	
btmpFPBrake :=  bBrakeStateOld <> vendorId;
bBrakeStateOld := vendorId;

mcReadDriveAddress(
	Axis:= Axis, 
	Execute:= btmpFPBrake, 
	Done=> , 
	Busy=> , 
	Error=> , 
	ErrorID=> , 
	DriveAddress=> Axis.DriveAddress);

	st_Trq_options.EnableManualTorqueStartValue :=TRUE;
	st_Trq_options.ManualTorqueStartValue:= 0.5;
	bTorqueReached:=fbAxisTorqueControl.InTorque;
	
fbAxisTorqueControl	(
	Axis:= Axis , 
	Execute:=bAxisMoveTorqueExecute , 
	Relative:= , 
	Torque:= 2 , 
	TorqueRamp:= 1, 
	VelocityLimitHigh:= 500, 
	VelocityLimitLow:= -500, 
	BufferMode:= , 
	Options:= ,//st_Trq_options , 
	InTorque=> , 
	Busy=> busy, 
	Active=> , 
	CommandAborted=> , 
	Error=> act, 
	ErrorId=> id );

//	fbEcCoeSdoRead(
//	sNetId:= Axis.DriveAddress.NetID,
//	nSlaveAddr:= Axis.DriveAddress.SlaveAddress,
//	nSubIndex:= 16#1, 
//	nIndex:= 16#8012, 
//	pDstBuf:= ADR(bBrakeStateOld), 
//	cbBufLen:= SIZEOF(bBrakeStateOld), 
//	bExecute:= mcReadDriveAddress.done, 
//	tTimeout:= , 
//	bBusy=> , 
//	bError=> , 
//	nErrId=> , 
//	cbRead=> );

fbEcCoeSdoWrite(
	sNetId:= Axis.DriveAddress.NetID,
	nSlaveAddr:= Axis.DriveAddress.SlaveAddress, 
	nSubIndex:= 16#1, 
	nIndex:= 16#8012, 
	pSrcBuf:= ADR(bBrakeStateOld), 
	cbBufLen:= SIZEOF(bBrakeStateOld), 
	bExecute:= mcReadDriveAddress.done, 
	tTimeout:= , 
	bBusy=> , 
	bError=> , 
	nErrId=> );
	
			IF bHardwareReset THEN
				FB_SoEReset(
				Axis:= Axis,	
				Execute:= TRUE,
				);
				IF NOT FB_SoEReset.Busy THEN
					FB_SoEReset(
					Axis:= Axis,	
					Execute:= FALSE,
					);
					bHardwareReset:= FALSE;
				END_IF	
			END_IF		

stManualModeAxis.actualPosition:=axis.NcToPlc.ActPos;
stManualModeAxis.actualVelocity:=axis.NcToPlc.ActVelo;
Actual_Torque:=fActualTorque;
//###################################################################################
//###################################################################################

//Output Signals
	sAxisState := TO_STRING(iSchritt);
	bAxisHomed := bAxisIsHomed;
	bAxisError := bAxisInError OR iSchritt = ENUM_Axis.Error;
	bAxis_ready := (iSchritt = ENUM_Axis.Ready);
	bAxisEnabled:= (iSchritt <> ENUM_Axis.PowerOFF) AND (iSchritt <> ENUM_Axis.Error);
	
IF In_range(stManualModeAxis.actualPosition,0,2) THEN
	baxis_in_home_pos:=TRUE;
ELSE
	baxis_in_home_pos:=FALSE;		
END_IF	
	
IF Safe_move_Conditions THEN
	bsafe_to_move:=TRUE;
	fOverride := 100;
ELSE
	bsafe_to_move:=FALSE;
	fOverride := 0;
END_IF	
IF bmove_home THEN
	CASE moving_home OF
		0:IF bmove_home AND bAxisEnabled AND NOT baxis_in_home_pos THEN
            fTargetPosition:=0;
			IF fTargetVelocity=0 THEN
				fTargetVelocity:=50;
			END_IF
		    moving_home:=1;	
		  ELSIF baxis_in_home_pos THEN
			bmove_home:=FALSE;
			moving_home:=0;		
		  END_IF
	   
		1: bMoveAbsolute:=TRUE; 
		  IF bMoveAbsolute THEN
			   moving_home:=2; 
		  END_IF
		   	
		2:  IF In_range(stManualModeAxis.actualPosition,0,1) OR fbAxisMoveAbsolute.Done THEN
			 //fbAxisMoveAbsolute.Execute:=FALSE;
			// moving_home:=0;
			 bmove_home:=FALSE;
		    END_IF		
	END_CASE
ELSE
	moving_home:=0;
END_IF	

Actual_position:=stManualModeAxis.actualPosition;
Actual_velocity:=stManualModeAxis.actualVelocity;

bAxisEnabled:= NOT bAxisError AND fbAxisPower.Status;



///////////////////////////////////// AUTO HOMING	////////////////////////////////
START_TIMER(IN:=bAxisPowerExecute , PT:=T#3S, Q=> , ET=> );
IF START_TIMER.Q THEN
	

bSet_Encoder_Zero:=NOT TRIAL OR home_pressed;

bSet_Encoder_Zero_Rtrig.CLK:=bSet_Encoder_Zero;
bSet_Encoder_Zero_Rtrig();

IF bSet_Encoder_Zero_Rtrig.Q THEN Step :=10; END_IF

CASE Step OF 
10:
	lrRead_set_Value:=0; lrWrite_set_Value:=0; bRead_set_Value:=FALSE; bWrite_set_Value :=FALSE; 
	Step:=Step+10;
20:
	lrWrite_set_Value:=0; bWrite_set_Value :=TRUE; 
	tDummy.IN:=TRUE;
	IF tDummy.Q THEN tDummy.IN:=FALSE ; bWrite_set_Value := FALSE;Step:= step+10; END_IF
30:	IF home_pressed THEN
	lrWrite_set_Value:= Axis.NcToPlc.ActPos * -1;
	ELSE
	 lrWrite_set_Value:=HOMING_VALUE;
	END_IF;
	Step:= step+10;
40:
	bWrite_set_Value := TRUE; tDummy.IN:=TRUE;
	IF tDummy.Q THEN tDummy.IN:=FALSE ;Step:= step+10; bWrite_set_Value := FALSE; END_IF
	IF ADSWRITE_Set_Val.ERR  THEN bWrite_set_Value := FALSE;tDummy.IN:=FALSE; Step:=10; END_IF
50:
	IF (LREAL_TO_INT(Axis.NcToPlc.ActPos*10)=0 OR (lrWrite_set_Value=HOMING_VALUE)) AND ( home_pressed OR NOT TRIAL) THEN
		bHome_ref_done:=TRUE;	step:=99; bSet_Encoder_Zero:=FALSE; 
	ELSE
 		step:=10;
END_IF 
	
END_CASE

FB_GetLocalAmsNetId_system.bExecute:=TRUE;
FB_GetLocalAmsNetId_system();

ADSWRITE_Set_Val(
	NETID:=FB_GetLocalAmsNetId_system.AddrString , 
	PORT:=501 , 	
	IDXGRP:=HME_WRITE_ADD, 	
	IDXOFFS:=16#07,  
	LEN:= SIZEOF(lrWrite_set_Value), 
	SRCADDR:= ADR(lrWrite_set_Value) , 
	WRITE:=bWrite_set_Value ,   	    
	TMOUT:=T#500MS , 
	BUSY=> ,  
	ERR=> , 	
	ERRID=> );	

tDummy.PT:=T#20MS;
tDummy();	
	
(*MC_Power1(
	Axis:=Axis, 
	Enable:=bEnable AND NOT home_pressed, 
	Enable_Positive:= 1, 
	Enable_Negative:= 1, 
	Override:=100 , 
	BufferMode:= , 
	Options:= , 
	Status=> , 
	Busy=> , 
	Active=> , 
	Error=> , 
	ErrorID=> );*)

TRIAL := (step=99);

IF (lrWrite_set_Value<>HOMING_VALUE)AND(step=99)THEN
	HOMING_VALUE:=lrWrite_set_Value;

END_IF	

IF step=99 THEN
	home_pressed:=FALSE;
 	bHome:=FALSE;
	bHomeDone := TRUE;
	//bHome := FALSE;
	stManualModeAxis.homing:= FALSE;
	//bAxisHomeExecute:= FALSE;
	//iSchritt := ENUM_Axis.Ready;	
END_IF
END_IF	
	
	
//############################		SERVO LIMIT 	##############################	

IF NOT LIMIT_BYPASS THEN

IF (stManualModeAxis.actualPosition>=Servo_Low_Limit) THEN
	LEG_LIMIT			:= TRUE;
ELSE	
	LEG_LIMIT			:= FALSE;
END_IF;

IF stManualModeAxis.actualPosition<=Servo_High_Limit THEN
	POS_LIMIT			:= TRUE;	
ELSE
	POS_LIMIT			:= FALSE;
END_IF
 
IF (fTargetPosition<=Servo_High_Limit) AND (fTargetPosition>=Servo_Low_Limit) THEN
	AUTO_TARGET_POSITION:=fTargetPosition;
ELSIF (fTargetPosition>=Servo_High_Limit)THEN
	AUTO_TARGET_POSITION:=Servo_High_Limit;
ELSIF (fTargetPosition<=Servo_Low_Limit) AND (fTargetPosition<=Servo_High_Limit) THEN
	AUTO_TARGET_POSITION:=Servo_Low_Limit;	
END_IF

IF (stManualModeAxis.targetPositon<=Servo_High_Limit) AND (stManualModeAxis.targetPositon>=Servo_Low_Limit) THEN
	MANUAL_TARGET_POSITION:=stManualModeAxis.targetPositon;
ELSIF (stManualModeAxis.targetPositon>=Servo_High_Limit)THEN
	MANUAL_TARGET_POSITION:=Servo_High_Limit;
ELSIF (stManualModeAxis.targetPositon<=Servo_Low_Limit) AND (stManualModeAxis.targetPositon<=Servo_High_Limit) THEN
	MANUAL_TARGET_POSITION:=Servo_Low_Limit;	
END_IF

IF (stManualModeAxis.actualPosition-WARNING_LIMIT)<=Servo_Low_Limit AND (stManualModeAxis.actualPosition+WARNING_LIMIT)<=Servo_High_Limit THEN
	SERVO_LIMIT_WARNING	:= TRUE;
ELSE
	SERVO_LIMIT_WARNING	:= FALSE;	
END_IF

ELSE	
	AUTO_TARGET_POSITION			:=fTargetPosition;
	MANUAL_TARGET_POSITION			:=stManualModeAxis.targetPositon;
END_IF

//################################			TORQUE LIMIT	############################

(*IF ((Torque_limit_perent=>0) AND (Torque_limit_perent<=100)) THEN
TORQUE_LIMIT	:= REAL_TO_UINT(327.68*Torque_limit_perent);	
END_IF*)

END_FUNCTION_BLOCK

// ---- POUs/Programs/OP10/OP10B_AUTO.TcPOU
PROGRAM OP10B_AUTO
VAR
	OP10B_ROBO_SYSTEM				: FB_Robot;
	OP10B_CYL_IP					: OP10_ORNG_CYL_IP;
	OP10B_CYL_OP					: OP10_ORNG_CYL_OP;
	OP10B_PNP_FB					: OP10_ORING_PNP;
	OP10B_ROBO_PNP_FB				: OP10_ROBO_PNP;
	OP10B_STN_MOVER					: INT;
	OP10B_OUT_ORNG_DN				: BOOL;
	OP10B_AGLE_LH_CMR_TRG			: BOOL;
	OP10B_AGLE_RH_CMR_TRG			: BOOL;	
	OP10B_RDY_TO_PLC_ORNG			: BOOL;
	OP10B_STN_ENABLE				: BOOL;
	OP10B_ROBO_INZI_DN				: BOOL;	
// TEMPER

	trial: BOOL;
	tmr: Ton;
	alll: BOOL;
	OP10B_PROCESS_DN: BOOL;
	OP10B_RESULT_UPDATE: INT;
	OP10B_PROCESS_DN_TRG: R_TRIG;
END_VAR

OP10B_PNP_FB(
	AUTO:= OP10B_AUTO_RUNNING OR OP10B_STEP_RUNNING, 
	MANUAL:= OP10B_MANUAL_SELECTED, 
	ERROR:= OP10B_ERR, 
	START_ENABLE:= OP10B_START_ENABLE, 
	ROBO_MVED_SFE:= NOT OP10B_Rbt_In_O_Ring_Zone , 
	LH_CMR_OK:= OP10B_LH_CMR_OK AND OP10B_ORNG_RDY_PCK, 
	LH_CMR_NOK:= OP10B_LH_CMR_NOK AND OP10B_ORNG_RDY_PCK, 
	RH_CMR_OK:= OP10B_RH_CMR_OK AND OP10B_ORNG_RDY_PCK, 
	RH_CMR_NOK:= OP10B_RH_CMR_NOK AND OP10B_ORNG_RDY_PCK, 
	ROBO_REACHED:= OP10B_RDY_TO_PLC_ORNG, 
	CYL_INPUTS:= OP10B_CYL_IP,
	CONTINOUS_CHECK := OP10B_CYL_PNP_CHECK, 
	DELY_TIME:= , 
	O_RING_PLCED=> OP10B_OUT_ORNG_DN, 
	RDY_TO_PICK_ORNG=> OP10B_CYL_RDY_TO_PLC, 
	LH_REJ_DONE=> , 
	RH_REJ_DONE=> , 
	CYL_OUTPUTS=> OP10B_CYL_OP,
	ORNG_PCK_FRM_CNVY := OP10B_ORNG_PCK_DN);

	

// OP10B AUTO LOGIC CYLINDERS MAPPING 

									(*SENSOR_I/P*)
	OP10B_CYL_IP.DEGREE_0				:=I10B_ORING_ROTRY_CYL_O_DEG_I1031_0;
	OP10B_CYL_IP.DEGREE_180				:=I10B_ORING_ROTRY_CYL_180_DEG_I1031_1;
    OP10B_CYL_IP.HORIZ_CYL_SNR1         :=I10B_ORING_HORZ_CYL_REV_I1031_2;
    OP10B_CYL_IP.HORIZ_CYL_SNR2         :=I10B_ORING_HORZ_CYL_FWD_I1031_3;
    OP10B_CYL_IP.LH_O_GRP_SNR1       	:=I10B_ORING_LH_GRPR_CLSE_I1030_2;
    OP10B_CYL_IP.LH_O_GRP_SNR2          :=I10B_ORING_LH_GRPR_OPN_I1030_3;
    OP10B_CYL_IP.LH_O_PUSH_SNR1         :=NOT I10B_ORING_LH_PUSHR_CYL_REV_I1030_4;
    OP10B_CYL_IP.LH_O_PUSH_SNR2         :=I10B_ORING_LH_PUSHR_CYL_REV_I1030_4;
    OP10B_CYL_IP.LH_REJ_SNR1            :=I10B_LH_FIRTRE_ORING_REJ_CYL_REV_I1031_6;
    OP10B_CYL_IP.LH_REJ_SNR2            :=I10B_LH_FIRTRE_ORING_REJ_CYL_FWD_I1031_7;
	OP10B_CYL_IP.RH_O_GRP_SNR1			:=I10B_ORING_RH_GRPR_CLSE_I1030_6 ;
    OP10B_CYL_IP.RH_O_GRP_SNR2          :=I10B_ORING_RH_GRPR_OPN_I1030_5;
    OP10B_CYL_IP.RH_O_PUSH_SNR1         :=NOT I10B_ORING_RH_PUSHR_CYL_REV_I1030_7;
    OP10B_CYL_IP.RH_O_PUSH_SNR2         :=I10B_ORING_RH_PUSHR_CYL_REV_I1030_7;
    OP10B_CYL_IP.RH_REJ_SNR1            :=I10B_RH_FIRTRE_ORING_REJ_CYL_REV_I1040_0;
    OP10B_CYL_IP.RH_REJ_SNR2            :=I10B_RH_FIRTRE_ORING_REJ_CYL_FWD_I1040_1;
    OP10B_CYL_IP.VERT_CYL_SNR1          :=I10B_ORING_VERT_CYL_UP_I1031_4;
    OP10B_CYL_IP.VERT_CYL_SNR2          :=I10B_ORING_VERT_CYL_DWN_I1031_5;
	
									(*CYLINDER_AUTO_O/P*)	
	
	OP10B_ALL_CYL_HOME_FB				:=OP10B_CYL_OP.ALL_HOME			;
	OP10B_O_0DEGRE_AUTOCMD1				:=OP10B_CYL_OP.DEGREE_AUT_CMD1	;
	OP10B_O_180DEGRE_AUTOCMD2   		:=OP10B_CYL_OP.DEGREE_AUT_CMD2    ;
	OP10B_O_HORZ_AUTOCMD1    			:=OP10B_CYL_OP.HORIZ_CYL_AUT_CMD1 ;
	OP10B_O_HORZ_AUTOCMD2    			:=OP10B_CYL_OP.HORIZ_CYL_AUT_CMD2 ;
	OP10B_A_O_LHGRIP_ONOFF    			:=OP10B_CYL_OP.LH_O_GRP_VALVE_ON  ;
	OP10B_A_O_LHPUSH_CYL    			:=OP10B_CYL_OP.LH_O_PSH_VALVE_ON  ;
	OP10B_A_O_RHGRIP_ONOFF    			:=OP10B_CYL_OP.RH_O_GRP_VALVE_ON  ;
	OP10B_A_O_RHPUSH_CYL    			:=OP10B_CYL_OP.RH_O_PSH_VALVE_ON  ;
	OP10B_O_VERT_AUTOCMD1    			:=OP10B_CYL_OP.VERT_CYL_AUT_CMD1  ;
	OP10B_O_VERT_AUTOCMD2    			:=OP10B_CYL_OP.VERT_CYL_AUT_CMD2  ;

//###############		ROBO	###################

OP10B_ROBO_PNP_FB(
	AUTO:= OP10B_AUTO_RUNNING OR OP10B_STEP_RUNNING, 
	MANUAL:= OP10B_MANUAL_SELECTED, 
	ERROR:= OP10B_ERR, 
	START_ENABLE:= OP10B_START_ENABLE, 
	ROBO_STATUS_FB:= OP10B_ROBO_STATUS, 
	ROBO_GRP_STUS:= OP10B_GRP_STATUS, 
	BDY1_RDY_PCK:=OP10_LH_CMP_RDY_PCK , 
	BDY2_RDY_PCK:=OP10_RH_CMP_RDY_PCK , 
	BDY1_PCK_BYPAS:= OP10B_BDY1_PCK_BYPAS, 
	BDY2_PCK_BYPAS:= OP10B_BDY2_PCK_BYPAS, 
	O_RNG_NEED:= , 
	PLC_OUTR_ORNG_DN:= OP10B_OUT_ORNG_DN OR trial, 
	CMR_RESULT_DN:= OP10B_CMR_DN_RSLT, 
	LH_CMR_ORNG_OK:= OP10B_LH_CMR_OK, 
	RH_CMR_ORING_OK:= OP10B_RH_CMR_OK,
	STN_ENABLE := OP10B_STN_ENABLE,
	OP10_STN_MOVER := OP10B_STN_MOVER,
	START_HOMING := OP10B_START_HOMNG,
	ROBO_IN_HOME := OP10B_Rbt_In_Home,
	STN_MOVER_NUM := OP10B_STN_MOVER,
	LH_BODY_GRIP_HME_DN := OP10B_SRV_LH_BDYGRP_CNT.Axis_In_Home,
	RH_BODY_GRIP_HME_DN := OP10B_SRV_RH_BDYGRP_CNT.Axis_In_Home,
	LH_BODY_ROTRY_HME_DN := OP10B_SRV_LH_BDYANG_CNT.Axis_In_Home,
	RH_BODY_ROTRY_HME_DN := OP10B_SRV_RH_BDYANG_CNT.Axis_In_Home,
	SEC_SING_CYL_SNR1 := OP10_BDY_SING_SEC.Sensor1,
	FRT_SING_CYL_SNR1 := OP10_BDY_SING_FRT.Sensor1,
	CMP_GRIPPED := OP10B_CMP_PRS_ROBO,
	ROBO_GRP_OPN := OP10B_ROBO_Gripper_Open,
	ROBO_IN_ORING_ZONE := OP10B_Rbt_In_O_Ring_Zone, 
	ROBO_CTRL_WRD=> OP10B_ROBO_CNTRL, 
	ROBO_GRP_CNTRL=> OP10B_GRP_CNTRL, 
	LH_CAMERA_TRIGGER=> OP10B_AGLE_LH_CMR_TRG, 
	RH_CAMERA_TRIGGER=> OP10B_AGLE_RH_CMR_TRG, 
	PLC_OUTR_ORNG=> OP10B_RDY_TO_PLC_ORNG,
	GRIPPER_HOME => OP10B_GRIPPER_HOME,
	OP10_CURR_MOVER => OP10B_CURR_MOVER,
	PROCESS_DONE := OP10B_PROCESS_DN,
	LH_PART_STATUS => ,
	RH_PART_STATUS => ,
	PROCESS_DONE => );

	OP10B_CMR_DN_RSLT			:= TRUE;						// should be deleted
	OP10B_LH_CMR_OK             := TRUE;						// should be deleted
	OP10B_RH_CMR_OK             := TRUE;						// should be deleted
	
(*tmr(IN:= OP10B_STN_ENABLE, PT:=T#10MS , Q=> , ET=> );
IF tmr.Q THEN
	IF (MOVER_CMP_STATUS[OP10B_STN_MOVER][1]=0) THEN
	MOVER_CMP_STATUS[OP10B_STN_MOVER][1] := 10;		
	END_IF
	IF (MOVER_CMP_STATUS[OP10B_STN_MOVER][2]=0) THEN
	MOVER_CMP_STATUS[OP10B_STN_MOVER][2] := 10;
	END_IF	
	ALL_STATION_DONE.POSITION_DONE[OP10B_XTS_POS_NO]:= TRUE;	
	END_IF*)

	(*IF  OP10B_PROCESS_DN THEN
	IF (MOVER_CMP_STATUS[OP10B_STN_MOVER][1]=0) THEN
	MOVER_CMP_STATUS[OP10B_CURR_MOVER][1] := OP10B_ROBO_PNP_FB.LH_PART_STATUS;		
	END_IF
	IF (MOVER_CMP_STATUS[OP10B_STN_MOVER][2]=0) THEN
	MOVER_CMP_STATUS[OP10B_CURR_MOVER][2] := OP10B_ROBO_PNP_FB.RH_PART_STATUS;
	END_IF	
	END_IF
	IF OP10B_PROCESS_DN AND (OP10B_CURR_MOVER = OP10B_STN_MOVER) AND (MOVER_CMP_STATUS[OP10B_STN_MOVER][1]=10 OR MOVER_CMP_STATUS[OP10B_STN_MOVER][1]=11) AND 
		(MOVER_CMP_STATUS[OP10B_STN_MOVER][2]=10 OR MOVER_CMP_STATUS[OP10B_STN_MOVER][2]=11) THEN
	STATION_DONE[OP10B_CURR_MOVER][OP10B_XTS_POS_NO]			:= TRUE;
	IF 	MOVER_STP_NO[OP10B_CURR_MOVER]<>((OP10B_XTS_POS_NO*10)+1) THEN
	OP10B_CURR_MOVER											:= 0;	
	OP10B_PROCESS_DN											:= FALSE;	
	END_IF
	END_IF*)
	
	
		CASE OP10B_RESULT_UPDATE OF
		0: IF OP10B_PROCESS_DN THEN
			OP10B_RESULT_UPDATE			:= 5;
		END_IF
		
		5: 	IF OP10B_PROCESS_DN THEN
			IF (MOVER_CMP_STATUS[OP10B_STN_MOVER][1]=0) THEN
			MOVER_CMP_STATUS[OP10B_CURR_MOVER][1] := OP10B_ROBO_PNP_FB.LH_PART_STATUS;		
			END_IF
			IF (MOVER_CMP_STATUS[OP10B_STN_MOVER][2]=0) THEN
			MOVER_CMP_STATUS[OP10B_CURR_MOVER][2] := OP10B_ROBO_PNP_FB.RH_PART_STATUS;
			END_IF		
			IF OP10B_PROCESS_DN AND (OP10B_CURR_MOVER = OP10B_STN_MOVER) AND (MOVER_CMP_STATUS[OP10B_STN_MOVER][1]=10 OR MOVER_CMP_STATUS[OP10B_STN_MOVER][1]=11) AND 
		(MOVER_CMP_STATUS[OP10B_STN_MOVER][2]=10 OR MOVER_CMP_STATUS[OP10B_STN_MOVER][2]=11) THEN
			OP10B_RESULT_UPDATE			:= 10;
			END_IF
			END_IF
	
		10:	STATION_DONE[OP10B_CURR_MOVER][OP10B_XTS_POS_NO]			:= TRUE;
			IF 	MOVER_STP_NO[OP10B_CURR_MOVER]<>((OP10B_XTS_POS_NO*10)+1)THEN
			OP10B_CURR_MOVER											:= 0;	
			OP10B_PROCESS_DN											:= FALSE;
			OP10B_RESULT_UPDATE											:= 15;
			END_IF
			
		15: OP10B_PROCESS_DN_TRG(CLK:= OP10B_PROCESS_DN, Q=> );
			IF OP10B_PROCESS_DN_TRG.Q THEN
			OP10B_RESULT_UPDATE											:= 0;	
			END_IF
	END_CASE

	
	
// ###########################			OP10B_ROBO_STATUS_CONTROL	####################################
	
	OP10B_ROBO_STATUS.BDY_PCK_POSITION	  		:= OP10B_ROBO_Gripper_Close AND OP10B_Rbt_In_Pick_Zone;//OP10B_Rbt_In_Pick_Zone
//	OP10B_ROBO_STATUS.BDY_S_PCK_POSITION		:= ;
	OP10B_ROBO_STATUS.BDY_CMR_CHK_POS		  	:= OP10B_Camera_Trigger; 							
//	OP10B_ROBO_STATUS.BDY_S_ORNG_POS		   	:= ;
	OP10B_ROBO_STATUS.BDY_ORNG_PLC_POS	  		:= OP10B_O_Ring_Pick_Pos_Reached AND OP10B_Rbt_In_O_Ring_Zone;//OP10B_Rbt_In_O_Ring_Zone
	OP10B_ROBO_STATUS.BDY_MVE_PLC_POS		  	:= OP10B_ROBO_Gripper_Open;//OP10B_Rbt_In_Place_Zone	
	OP10B_ROBO_STATUS.ROBO_SAFE_POS		    	:= NOT OP10B_Rbt_In_Place_Zone;
	OP10B_ROBO_STATUS.ROBO_REJ_POS				:= OP10B_Rbt_In_Reject_Zone;


	
	OP10B_A_BODY_READY_TO_PICK					:= 	OP10B_ROBO_CNTRL.BDY_PCK_POSITION	;	
//	                                      	 	:=  OP10B_ROBO_CNTRL.BDY_S_PCK_POSITION;	    
	OP10B_A_PICK_PART_OK                   		:=  OP10B_ROBO_CNTRL.BDY_CMR_CHK_POS		;
//					                      		:= 	OP10B_ROBO_CNTRL.BDY_S_ORNG_POS		;    
	OP10B_A_CAMERA_OK                      		:= 	OP10B_ROBO_CNTRL.BDY_ORNG_PLC_POS OR OP10B_ROBO_CNTRL.BDY_MVE_PLC_POS;    
//	                                       		:= 	OP10B_ROBO_CNTRL.ROBO_SAFE_POS		;    
//	                                       		:= 	OP10B_ROBO_CNTRL.ROBO_REJ_POS		;   


//##############################	OP10_GRP_STATUS_CONTROL	################################################

	OP10B_GRP_STATUS.LH_BDY_GRP_WRK_FB			:= OP10B_A_SRV_LH_GRPWRK_FB	;
	OP10B_GRP_STATUS.LH_BDY_GRP_HOM_FB		    := OP10B_A_SRV_LH_GRPHME_FB	;
	OP10B_GRP_STATUS.RH_BDY_GRP_WRK_FB		    := OP10B_A_SRV_RH_GRPWRK_FB	;
	OP10B_GRP_STATUS.RH_BDY_GRP_HME_FB		    := OP10B_A_SRV_RH_GRPHME_FB	;
	OP10B_GRP_STATUS.LH_BDY_ROTRY_WRK_FB		:= OP10B_SRV_LH_BDYANG_WRK_FB;
	OP10B_GRP_STATUS.LH_BDY_ROTRY_HOM_FB		:= OP10B_SRV_LH_BDYANG_HME_FB;
	OP10B_GRP_STATUS.RH_BDY_ROTRY_HME_FB		:= OP10B_SRV_RH_BDYANG_HME_FB;
	OP10B_GRP_STATUS.RH_BDY_ROTRY_WRK_FB		:= OP10B_SRV_RH_BDYANG_WRK_FB;
	OP10B_GRP_STATUS.RH_BDY_ROTRY_ZERO_FB		:= OP10B_SRV_RH_BDYANG_ZERO_FB;
	OP10B_GRP_STATUS.LH_BDY_ROTRY_ZERO_FB		:= OP10B_SRV_LH_BDYANG_ZERO_FB;
	OP10B_GRP_STATUS.RH_BDY_ROTRY_CMR_FB		:= OP10B_SRV_RH_BDYANG_CMR_FB;
	OP10B_GRP_STATUS.RH_BDY_RTRY_FITEE_FB		:= OP10B_SRV_RH_BDYANG_FITRE_FB;
	OP10B_GRP_STATUS.LH_BDY_ROTRY_CMR_FB		:= OP10B_SRV_LH_BDYANG_CMR_FB;	
	OP10B_GRP_STATUS.LH_BDY_RTRY_FITEE_FB		:= OP10B_SRV_LH_BDYANG_FITRE_FB;

	
	OP10B_A_SRV_LH_GRPWRK						:= OP10B_GRP_CNTRL.LH_BODY_GRIP_WRK	;
	OP10B_A_SRV_LH_GRPHME	        			:= OP10B_GRP_CNTRL.LH_BODY_GRIP_HOM	;
	OP10B_A_SRV_RH_GRPWRK	        			:= OP10B_GRP_CNTRL.RH_BODY_GRIP_WRK	;
	OP10B_A_SRV_RH_GRPHME	        			:= OP10B_GRP_CNTRL.RH_BODY_GRIP_HME	;
	OP10B_SRV_LH_BDYANG_WRK	        			:= OP10B_GRP_CNTRL.LH_BODY_ROTRY_WRK;	
	OP10B_SRV_LH_BDYANG_HME	        			:= OP10B_GRP_CNTRL.LH_BODY_ROTRY_HOM ;	
	OP10B_SRV_RH_BDYANG_WRK	        			:= OP10B_GRP_CNTRL.RH_BODY_ROTRY_WRK;	
	OP10B_SRV_RH_BDYANG_HME	        			:= OP10B_GRP_CNTRL.RH_BODY_ROTRY_HME ;	
	OP10B_SRV_LH_BDYANG_CMR						:= OP10B_GRP_CNTRL.LH_BODY_ROTRY_CMR;
	OP10B_SRV_LH_BDYANG_FITRE					:= OP10B_GRP_CNTRL.LH_BODY_RTRY_FITEE;	
	OP10B_SRV_RH_BDYANG_CMR						:= OP10B_GRP_CNTRL.RH_BODY_ROTRY_CMR;
	OP10B_SRV_RH_BDYANG_FITRE					:= OP10B_GRP_CNTRL.RH_BODY_RTRY_FITEE;
	
	
// STEPPER_NEGATIVE_HOME_METHOD
	
	OP10B_SRV_LH_BDYGRP_CNT.Axis_Home_Cmd		:=	OP10B_GRP_CNTRL.LH_BODY_GRIP_HOMING_1 ;
	OP10B_SRV_RH_BDYGRP_CNT.Axis_Home_Cmd	    :=	OP10B_GRP_CNTRL.RH_BODY_GRIP_HOMING_1 ;
	OP10B_SRV_LH_BDYANG_CNT.Axis_Home_Cmd	    :=	OP10B_GRP_CNTRL.LH_BODY_ROTRY_HOMING_1;
	OP10B_SRV_RH_BDYANG_CNT.Axis_Home_Cmd	    :=	OP10B_GRP_CNTRL.RH_BODY_ROTRY_HOMING_1;


//#####################################	ROBO_FB	####################################	                                               

OP10B_ROBO_SYSTEM(
	i_b_Operation_Enable_Feedback:= OP10B_Auto_Operation_Enable, 
	i_b_Auto_Enable_Feedback:= OP10B_Mirror_Auto_enable, 
	i_b_Servo_On_Feedback:= OP10B_Servo_ON_OFF_Status, 
	i_b_Servo_Off_Feedback:= OP10B_Mirror_SRVO_Off, 
	i_b_Error_Feedback:= OP10B_H_Error OR OP10B_L_Error, 
	i_b_Program_Start_Enable_Feedback:= OP10B_Program_Execute, 
	i_b_Robo_Stopping_Feedback:= OP10B_Program_Waiting, 
	i_b_Emergency_Pressed_Feedback:= OP10B_During_EMG_Stop, 
	i_b_Auto_Mode_Feedback:= OP10B_Mirror_Auto_enable, 
	i_b_Reset:= Servo_Reset, 
	i_b_RobotAutoManual:= OP10B_AUTO_SELECTED OR OP10B_STEP_SELECTED OR OP10B_MANUAL_SELECTED, 
	i_b_ProgramReset:= OP10B_ROBO_PRGM_RST, 
	o_b_Operation_Enable_Cmd=> OP10B_Operation_Enable, 
	o_b_Auto_Enable_Cmd=> OP10B_Auto_Enable, 
	o_b_Servo_On_Cmd=> OP10B_Servo_ON, 
	o_b_Servo_Off_Cmd=> OP10B_SERVO_OFF, 
	o_b_Error_Reset_Cmd=> OP10B_ERR_RST, 
	o_b_Program_Reset_Cmd=> OP10B_PRGM_RST, 
	o_b_Program_Start_Cmd=> OP10B_Start, 
	o_b_Program_Stop_Cmd=> OP10B_Stop , 
	o_b_RobotAutoManual=> , 
	o_b_Error=> );	
	
	OP10B_STOP2:=OP10B_Stop;
	WITH_ORING_VARIIENT			:= TRUE; 


/////////////////////////////////////////	OP10B_ROBO	////////////////////////////////////////////////////

	IF (MANUAL_SELECTED AND OP10B_M_BODY_READY_TO_PICK) OR 
		(OP10B_A_BODY_READY_TO_PICK AND NOT OP10A_BODY_READY_TO_PICK AND NOT OP10A_Rbt_In_Pick_Zone )THEN
		OP10B_BODY_READY_TO_PICK						:= TRUE;// BODY COMPONENT READY;
		OP10B_Pick_Zone_Safe							:= (OP10B_A_SRV_LH_GRPHME_FB OR OP10B_BDY1_PCK_BYPAS) AND 
															(OP10B_A_SRV_RH_GRPHME_FB OR OP10B_BDY2_PCK_BYPAS) AND 
															(OP10B_SRV_LH_BDYANG_HME OR OP10B_BDY1_PCK_BYPAS) AND 
															(OP10B_SRV_RH_BDYANG_HME OR OP10B_BDY2_PCK_BYPAS) AND 
																OP10_LH_CMP_RDY_PCK AND OP10_RH_CMP_RDY_PCK;			
	ELSE
		OP10B_BODY_READY_TO_PICK						:= FALSE;
		OP10B_Pick_Zone_Safe							:= FALSE;					
	END_IF

